LIN {X 0,Y 474.641,Z 374.861,A -85,B 0,C 180,E1 -7413.984,E2 -7413.984} C_VEL
LIN {X 0,Y 474.578,Z 374.865,A -85,B 0,C 180,E1 -7416.9,E2 -7416.9} C_VEL
LIN {X 0,Y 474.63,Z 374.866,A -85,B 0,C 180,E1 -7419.648,E2 -7419.648} C_VEL
LIN {X 0,Y 474.638,Z 374.859,A -85,B 0,C 180,E1 -7422.932,E2 -7422.932} C_VEL
LIN {X 0,Y 474.612,Z 374.864,A -85,B 0,C 180,E1 -7425.895,E2 -7425.895} C_VEL
LIN {X 0,Y 474.63,Z 374.861,A -85,B 0,C 180,E1 -7429.041,E2 -7429.041} C_VEL
LIN {X 0,Y 474.613,Z 374.865,A -85,B 0,C 180,E1 -7431.704,E2 -7431.704} C_VEL
LIN {X 0,Y 474.633,Z 374.859,A -85,B 0,C 180,E1 -7434.726,E2 -7434.726} C_VEL
LIN {X 0,Y 474.638,Z 374.86,A -85,B 0,C 180,E1 -7437.788,E2 -7437.788} C_VEL
LIN {X 0,Y 474.627,Z 374.862,A -85,B 0,C 180,E1 -7440.885,E2 -7440.885} C_VEL
LIN {X 0,Y 474.663,Z 374.859,A -85,B 0,C 180,E1 -7443.629,E2 -7443.629} C_VEL
LIN {X 0,Y 474.638,Z 374.864,A -85,B 0,C 180,E1 -7446.642,E2 -7446.642} C_VEL
LIN {X 0,Y 474.644,Z 374.992,A -85,B 0,C 180,E1 -7447.845,E2 -7447.845} C_VEL
LIN {X 0,Y 475.969,Z 382.275,A -85,B 0,C 180,E1 -7449.471,E2 -7449.471} C_VEL
LIN {X 0,Y 475.834,Z 390.327,A -85,B 0,C 180,E1 -7451.163,E2 -7451.163} C_VEL
LIN {X 0,Y 475.06,Z 393.516,A -85,B 0,C 180,E1 -7451.731,E2 -7451.731} C_VEL
LIN {X 0,Y 472.954,Z 398.571,A -85,B 0,C 180,E1 -7452.388,E2 -7452.388} C_VEL
LIN {X 0,Y 470.99,Z 404.444,A -85,B 0,C 180,E1 -7452.913,E2 -7452.913} C_VEL
LIN {X 0,Y 470.407,Z 409.431,A -85,B 0,C 180,E1 -7453.202,E2 -7453.202} C_VEL
LIN {X 0,Y 470.813,Z 412.936,A -85,B 0,C 180,E1 -7453.324,E2 -7453.324} C_VEL
LIN {X 0,Y 471.386,Z 416.146,A -85,B 0,C 180,E1 -7453.395,E2 -7453.395} C_VEL
LIN {X 0,Y 470.721,Z 508.175,A -85,B 0,C 180,E1 -7454.826,E2 -7454.826} C_VEL
LIN {X 0,Y 470.324,Z 521.294,A -85,B 0,C 180,E1 -7455.201,E2 -7455.201} C_VEL
LIN {X 0,Y 469.941,Z 533.362,A -85,B 0,C 180,E1 -7455.714,E2 -7455.714} C_VEL
LIN {X 0,Y 469.543,Z 544.921,A -85,B 0,C 180,E1 -7456.377,E2 -7456.377} C_VEL
LIN {X 0,Y 469.092,Z 556.415,A -85,B 0,C 180,E1 -7457.233,E2 -7457.233} C_VEL
LIN {X 0,Y 468.56,Z 566.889,A -85,B 0,C 180,E1 -7458.208,E2 -7458.208} C_VEL
LIN {X 0,Y 468.137,Z 575.446,A -85,B 0,C 180,E1 -7459.184,E2 -7459.184} C_VEL
LIN {X 0,Y 467.72,Z 583.328,A -85,B 0,C 180,E1 -7460.268,E2 -7460.268} C_VEL
LIN {X 0,Y 467.35,Z 591.034,A -85,B 0,C 180,E1 -7461.569,E2 -7461.569} C_VEL
LIN {X 0,Y 467.003,Z 598.104,A -85,B 0,C 180,E1 -7463.085,E2 -7463.085} C_VEL
LIN {X 0,Y 466.918,Z 602.812,A -85,B 0,C 180,E1 -7464.385,E2 -7464.385} C_VEL
LIN {X 0,Y 466.744,Z 606.42,A -85,B 0,C 180,E1 -7465.682,E2 -7465.682} C_VEL
LIN {X 0,Y 466.768,Z 608.283,A -85,B 0,C 180,E1 -7466.547,E2 -7466.547} C_VEL
LIN {X 0,Y 466.683,Z 609.689,A -85,B 0,C 180,E1 -7467.411,E2 -7467.411} C_VEL
LIN {X 0,Y 466.62,Z 611.305,A -85,B 0,C 180,E1 -7469.137,E2 -7469.137} C_VEL
LIN {X 0,Y 466.599,Z 611.541,A -85,B 0,C 180,E1 -7470,E2 -7470} C_VEL
LIN {X 0,Y 466.62,Z 611.354,A -85,B 0,C 180,E1 -7470.863,E2 -7470.863} C_VEL
LIN {X 0,Y 466.684,Z 609.803,A -85,B 0,C 180,E1 -7472.59,E2 -7472.59} C_VEL
LIN {X 0,Y 466.767,Z 608.446,A -85,B 0,C 180,E1 -7473.453,E2 -7473.453} C_VEL
LIN {X 0,Y 466.731,Z 605.582,A -85,B 0,C 180,E1 -7474.751,E2 -7474.751} C_VEL
LIN {X 0,Y 466.97,Z 601.692,A -85,B 0,C 180,E1 -7476.048,E2 -7476.048} C_VEL
LIN {X 0,Y 467.099,Z 596.678,A -85,B 0,C 180,E1 -7477.348,E2 -7477.348} C_VEL
LIN {X 0,Y 467.365,Z 590.367,A -85,B 0,C 180,E1 -7478.649,E2 -7478.649} C_VEL
LIN {X 0,Y 467.731,Z 582.464,A -85,B 0,C 180,E1 -7479.951,E2 -7479.951} C_VEL
LIN {X 0,Y 468.241,Z 572.632,A -85,B 0,C 180,E1 -7481.252,E2 -7481.252} C_VEL
LIN {X 0,Y 468.788,Z 562.317,A -85,B 0,C 180,E1 -7482.336,E2 -7482.336} C_VEL
LIN {X 0,Y 469.277,Z 550.683,A -85,B 0,C 180,E1 -7483.312,E2 -7483.312} C_VEL
LIN {X 0,Y 469.761,Z 539.099,A -85,B 0,C 180,E1 -7484.071,E2 -7484.071} C_VEL
LIN {X 0,Y 470.194,Z 527.053,A -85,B 0,C 180,E1 -7484.665,E2 -7484.665} C_VEL
LIN {X 0,Y 470.525,Z 513.933,A -85,B 0,C 180,E1 -7485.125,E2 -7485.125} C_VEL
LIN {X 0,Y 470.775,Z 501.287,A -85,B 0,C 180,E1 -7485.394,E2 -7485.394} C_VEL
LIN {X 0,Y 471.261,Z 415.355,A -85,B 0,C 180,E1 -7486.713,E2 -7486.713} C_VEL
LIN {X 0,Y 468.483,Z 400.834,A -85,B 0,C 180,E1 -7487.055,E2 -7487.055} C_VEL
LIN {X 0,Y 469.089,Z 386.049,A -85,B 0,C 180,E1 -7490.157,E2 -7490.157} C_VEL
LIN {X 0,Y 468.789,Z 381.795,A -85,B 0,C 180,E1 -7491.088,E2 -7491.088} C_VEL
LIN {X 0,Y 467.605,Z 375.744,A -85,B 0,C 180,E1 -7492.478,E2 -7492.478} C_VEL
LIN {X 0,Y 467.614,Z 375.739,A -85,B 0,C 180,E1 -7495.84,E2 -7495.84} C_VEL
LIN {X 0,Y 467.581,Z 375.744,A -85,B 0,C 180,E1 -7498.75,E2 -7498.75} C_VEL
LIN {X 0,Y 467.587,Z 375.736,A -85,B 0,C 180,E1 -7501.74,E2 -7501.74} C_VEL
LIN {X 0,Y 467.57,Z 375.745,A -85,B 0,C 180,E1 -7504.833,E2 -7504.833} C_VEL
LIN {X 0,Y 467.569,Z 375.739,A -85,B 0,C 180,E1 -7508.045,E2 -7508.045} C_VEL
LIN {X 0,Y 467.582,Z 375.737,A -85,B 0,C 180,E1 -7511.277,E2 -7511.277} C_VEL
LIN {X 0,Y 467.558,Z 375.74,A -85,B 0,C 180,E1 -7513.821,E2 -7513.821} C_VEL
LIN {X 0,Y 467.574,Z 375.742,A -85,B 0,C 180,E1 -7516.257,E2 -7516.257} C_VEL
LIN {X 0,Y 467.586,Z 375.741,A -85,B 0,C 180,E1 -7518.723,E2 -7518.723} C_VEL
LIN {X 0,Y 467.569,Z 375.74,A -85,B 0,C 180,E1 -7521.956,E2 -7521.956} C_VEL
LIN {X 0,Y 467.568,Z 375.738,A -85,B 0,C 180,E1 -7525.168,E2 -7525.168} C_VEL
LIN {X 0,Y 467.588,Z 375.743,A -85,B 0,C 180,E1 -7528.26,E2 -7528.26} C_VEL
LIN {X 0,Y 467.582,Z 375.736,A -85,B 0,C 180,E1 -7531.251,E2 -7531.251} C_VEL
LIN {X 0,Y 467.618,Z 375.732,A -85,B 0,C 180,E1 -7533.2,E2 -7533.2} C_VEL
LIN {X 0,Y 467.596,Z 375.739,A -85,B 0,C 180,E1 -7536.469,E2 -7536.469} C_VEL
LIN {X 0,Y 467.63,Z 375.734,A -85,B 0,C 180,E1 -7539.777,E2 -7539.777} C_VEL
LIN {X 0,Y 467.615,Z 375.735,A -85,B 0,C 180,E1 -7542.507,E2 -7542.507} C_VEL
LIN {X 0,Y 467.612,Z 375.733,A -85,B 0,C 180,E1 -7545.197,E2 -7545.197} C_VEL
LIN {X 0,Y 467.662,Z 375.732,A -85,B 0,C 180,E1 -7547.855,E2 -7547.855} C_VEL
LIN {X 0,Y 467.686,Z 375.725,A -85,B 0,C 180,E1 -7551.357,E2 -7551.357} C_VEL
LIN {X 0,Y 467.749,Z 375.723,A -85,B 0,C 180,E1 -7553.963,E2 -7553.963} C_VEL
LIN {X 0,Y 467.865,Z 375.704,A -85,B 0,C 180,E1 -7557.417,E2 -7557.417} C_VEL
LIN {X 0,Y 467.888,Z 375.704,A -85,B 0,C 180,E1 -7560,E2 -7560} C_VEL
LIN {X 0,Y 467.865,Z 375.701,A -85,B 0,C 180,E1 -7562.583,E2 -7562.583} C_VEL
LIN {X 0,Y 467.748,Z 375.72,A -85,B 0,C 180,E1 -7566.037,E2 -7566.037} C_VEL
LIN {X 0,Y 467.674,Z 375.725,A -85,B 0,C 180,E1 -7568.643,E2 -7568.643} C_VEL
LIN {X 0,Y 467.689,Z 375.725,A -85,B 0,C 180,E1 -7572.145,E2 -7572.145} C_VEL
LIN {X 0,Y 467.655,Z 375.731,A -85,B 0,C 180,E1 -7575.885,E2 -7575.885} C_VEL
LIN {X 0,Y 467.629,Z 375.736,A -85,B 0,C 180,E1 -7579.308,E2 -7579.308} C_VEL
LIN {X 0,Y 467.539,Z 375.743,A -85,B 0,C 180,E1 -7582.074,E2 -7582.074} C_VEL
LIN {X 0,Y 467.59,Z 375.737,A -85,B 0,C 180,E1 -7584.888,E2 -7584.888} C_VEL
LIN {X 0,Y 467.625,Z 375.734,A -85,B 0,C 180,E1 -7587.769,E2 -7587.769} C_VEL
LIN {X 0,Y 467.572,Z 375.742,A -85,B 0,C 180,E1 -7591.045,E2 -7591.045} C_VEL
LIN {X 0,Y 467.581,Z 375.736,A -85,B 0,C 180,E1 -7594.24,E2 -7594.24} C_VEL
LIN {X 0,Y 467.552,Z 375.748,A -85,B 0,C 180,E1 -7597.186,E2 -7597.186} C_VEL
LIN {X 0,Y 467.578,Z 375.737,A -85,B 0,C 180,E1 -7600.265,E2 -7600.265} C_VEL
LIN {X 0,Y 467.59,Z 375.737,A -85,B 0,C 180,E1 -7602.567,E2 -7602.567} C_VEL
LIN {X 0,Y 467.575,Z 375.745,A -85,B 0,C 180,E1 -7605.053,E2 -7605.053} C_VEL
LIN {X 0,Y 467.592,Z 375.738,A -85,B 0,C 180,E1 -7607.44,E2 -7607.44} C_VEL
LIN {X 0,Y 467.586,Z 375.742,A -85,B 0,C 180,E1 -7610.855,E2 -7610.855} C_VEL
LIN {X 0,Y 467.564,Z 375.739,A -85,B 0,C 180,E1 -7614.261,E2 -7614.261} C_VEL
LIN {X 0,Y 467.585,Z 375.739,A -85,B 0,C 180,E1 -7617.321,E2 -7617.321} C_VEL
LIN {X 0,Y 467.574,Z 375.745,A -85,B 0,C 180,E1 -7620.667,E2 -7620.667} C_VEL
LIN {X 0,Y 467.62,Z 375.738,A -85,B 0,C 180,E1 -7623.2,E2 -7623.2} C_VEL
LIN {X 0,Y 467.656,Z 375.805,A -85,B 0,C 180,E1 -7624.532,E2 -7624.532} C_VEL
LIN {X 0,Y 469.817,Z 387.641,A -85,B 0,C 180,E1 -7626.879,E2 -7626.879} C_VEL
LIN {X 0,Y 469.192,Z 401.354,A -85,B 0,C 180,E1 -7629.39,E2 -7629.39} C_VEL
LIN {X 0,Y 468.532,Z 417.506,A -85,B 0,C 180,E1 -7632.317,E2 -7632.317} C_VEL
LIN {X 0,Y 468.356,Z 421.166,A -85,B 0,C 180,E1 -7632.978,E2 -7632.978} C_VEL
LIN {X 0,Y 471.298,Z 439.48,A -85,B 0,C 180,E1 -7633.378,E2 -7633.378} C_VEL
LIN {X 0,Y 470.596,Z 529.173,A -85,B 0,C 180,E1 -7634.766,E2 -7634.766} C_VEL
LIN {X 0,Y 470.239,Z 542.449,A -85,B 0,C 180,E1 -7635.143,E2 -7635.143} C_VEL
LIN {X 0,Y 469.768,Z 554.613,A -85,B 0,C 180,E1 -7635.653,E2 -7635.653} C_VEL
LIN {X 0,Y 469.294,Z 566.886,A -85,B 0,C 180,E1 -7636.357,E2 -7636.357} C_VEL
LIN {X 0,Y 468.767,Z 578.482,A -85,B 0,C 180,E1 -7637.224,E2 -7637.224} C_VEL
LIN {X 0,Y 468.291,Z 588.923,A -85,B 0,C 180,E1 -7638.201,E2 -7638.201} C_VEL
LIN {X 0,Y 467.866,Z 597.459,A -85,B 0,C 180,E1 -7639.177,E2 -7639.177} C_VEL
LIN {X 0,Y 467.468,Z 605.335,A -85,B 0,C 180,E1 -7640.262,E2 -7640.262} C_VEL
LIN {X 0,Y 467.123,Z 613.026,A -85,B 0,C 180,E1 -7641.565,E2 -7641.565} C_VEL
LIN {X 0,Y 466.86,Z 620.118,A -85,B 0,C 180,E1 -7643.083,E2 -7643.083} C_VEL
LIN {X 0,Y 466.784,Z 624.837,A -85,B 0,C 180,E1 -7644.384,E2 -7644.384} C_VEL
LIN {X 0,Y 466.647,Z 628.44,A -85,B 0,C 180,E1 -7645.681,E2 -7645.681} C_VEL
LIN {X 0,Y 466.661,Z 630.3,A -85,B 0,C 180,E1 -7646.546,E2 -7646.546} C_VEL
LIN {X 0,Y 466.66,Z 631.695,A -85,B 0,C 180,E1 -7647.41,E2 -7647.41} C_VEL
LIN {X 0,Y 466.589,Z 633.296,A -85,B 0,C 180,E1 -7649.137,E2 -7649.137} C_VEL
LIN {X 0,Y 466.598,Z 633.513,A -85,B 0,C 180,E1 -7650,E2 -7650} C_VEL
LIN {X 0,Y 466.607,Z 632.691,A -85,B 0,C 180,E1 -7651.726,E2 -7651.726} C_VEL
LIN {X 0,Y 466.66,Z 631.698,A -85,B 0,C 180,E1 -7652.589,E2 -7652.589} C_VEL
LIN {X 0,Y 466.661,Z 630.304,A -85,B 0,C 180,E1 -7653.453,E2 -7653.453} C_VEL
LIN {X 0,Y 466.692,Z 627.372,A -85,B 0,C 180,E1 -7654.751,E2 -7654.751} C_VEL
LIN {X 0,Y 466.779,Z 623.403,A -85,B 0,C 180,E1 -7656.05,E2 -7656.05} C_VEL
LIN {X 0,Y 466.978,Z 617.299,A -85,B 0,C 180,E1 -7657.567,E2 -7657.567} C_VEL
LIN {X 0,Y 467.232,Z 610.628,A -85,B 0,C 180,E1 -7658.869,E2 -7658.869} C_VEL
LIN {X 0,Y 467.59,Z 602.351,A -85,B 0,C 180,E1 -7660.172,E2 -7660.172} C_VEL
LIN {X 0,Y 468.057,Z 593.87,A -85,B 0,C 180,E1 -7661.256,E2 -7661.256} C_VEL
LIN {X 0,Y 468.583,Z 583.778,A -85,B 0,C 180,E1 -7662.304,E2 -7662.304} C_VEL
LIN {X 0,Y 468.97,Z 573.014,A -85,B 0,C 180,E1 -7663.211,E2 -7663.211} C_VEL
LIN {X 0,Y 469.484,Z 561.645,A -85,B 0,C 180,E1 -7663.968,E2 -7663.968} C_VEL
LIN {X 0,Y 469.931,Z 549.982,A -85,B 0,C 180,E1 -7664.563,E2 -7664.563} C_VEL
LIN {X 0,Y 470.365,Z 537.457,A -85,B 0,C 180,E1 -7665.019,E2 -7665.019} C_VEL
LIN {X 0,Y 470.637,Z 524.776,A -85,B 0,C 180,E1 -7665.315,E2 -7665.315} C_VEL
LIN {X 0,Y 471.121,Z 438.262,A -85,B 0,C 180,E1 -7666.646,E2 -7666.646} C_VEL
LIN {X 0,Y 468.379,Z 421.186,A -85,B 0,C 180,E1 -7667.014,E2 -7667.014} C_VEL
LIN {X 0,Y 469.104,Z 403.829,A -85,B 0,C 180,E1 -7670.156,E2 -7670.156} C_VEL
LIN {X 0,Y 469.829,Z 388.878,A -85,B 0,C 180,E1 -7672.888,E2 -7672.888} C_VEL
LIN {X 0,Y 469.111,Z 383.371,A -85,B 0,C 180,E1 -7673.953,E2 -7673.953} C_VEL
LIN {X 0,Y 467.646,Z 375.734,A -85,B 0,C 180,E1 -7675.52,E2 -7675.52} C_VEL
LIN {X 0,Y 467.63,Z 375.736,A -85,B 0,C 180,E1 -7677.768,E2 -7677.768} C_VEL
LIN {X 0,Y 467.572,Z 375.745,A -85,B 0,C 180,E1 -7681.045,E2 -7681.045} C_VEL
LIN {X 0,Y 467.591,Z 375.735,A -85,B 0,C 180,E1 -7684.242,E2 -7684.242} C_VEL
LIN {X 0,Y 467.55,Z 375.746,A -85,B 0,C 180,E1 -7687.186,E2 -7687.186} C_VEL
LIN {X 0,Y 467.579,Z 375.737,A -85,B 0,C 180,E1 -7690.264,E2 -7690.264} C_VEL
LIN {X 0,Y 467.588,Z 375.739,A -85,B 0,C 180,E1 -7692.567,E2 -7692.567} C_VEL
LIN {X 0,Y 467.573,Z 375.744,A -85,B 0,C 180,E1 -7695.053,E2 -7695.053} C_VEL
LIN {X 0,Y 467.591,Z 375.737,A -85,B 0,C 180,E1 -7697.44,E2 -7697.44} C_VEL
LIN {X 0,Y 467.584,Z 375.744,A -85,B 0,C 180,E1 -7700.855,E2 -7700.855} C_VEL
LIN {X 0,Y 467.562,Z 375.741,A -85,B 0,C 180,E1 -7704.261,E2 -7704.261} C_VEL
LIN {X 0,Y 467.584,Z 375.737,A -85,B 0,C 180,E1 -7707.321,E2 -7707.321} C_VEL
LIN {X 0,Y 467.573,Z 375.746,A -85,B 0,C 180,E1 -7710.667,E2 -7710.667} C_VEL
LIN {X 0,Y 467.615,Z 375.734,A -85,B 0,C 180,E1 -7713.2,E2 -7713.2} C_VEL
LIN {X 0,Y 467.593,Z 375.742,A -85,B 0,C 180,E1 -7716.469,E2 -7716.469} C_VEL
LIN {X 0,Y 467.627,Z 375.731,A -85,B 0,C 180,E1 -7719.777,E2 -7719.777} C_VEL
LIN {X 0,Y 467.61,Z 375.741,A -85,B 0,C 180,E1 -7722.507,E2 -7722.507} C_VEL
LIN {X 0,Y 467.609,Z 375.733,A -85,B 0,C 180,E1 -7725.197,E2 -7725.197} C_VEL
LIN {X 0,Y 467.686,Z 375.725,A -85,B 0,C 180,E1 -7727.855,E2 -7727.855} C_VEL
LIN {X 0,Y 467.673,Z 375.725,A -85,B 0,C 180,E1 -7731.357,E2 -7731.357} C_VEL
LIN {X 0,Y 467.74,Z 375.72,A -85,B 0,C 180,E1 -7733.963,E2 -7733.963} C_VEL
LIN {X 0,Y 467.862,Z 375.702,A -85,B 0,C 180,E1 -7737.417,E2 -7737.417} C_VEL
LIN {X 0,Y 467.886,Z 375.704,A -85,B 0,C 180,E1 -7740,E2 -7740} C_VEL
LIN {X 0,Y 467.863,Z 375.704,A -85,B 0,C 180,E1 -7742.583,E2 -7742.583} C_VEL
LIN {X 0,Y 467.747,Z 375.723,A -85,B 0,C 180,E1 -7746.037,E2 -7746.037} C_VEL
LIN {X 0,Y 467.683,Z 375.725,A -85,B 0,C 180,E1 -7748.643,E2 -7748.643} C_VEL
LIN {X 0,Y 467.659,Z 375.733,A -85,B 0,C 180,E1 -7752.145,E2 -7752.145} C_VEL
LIN {X 0,Y 467.642,Z 375.733,A -85,B 0,C 180,E1 -7755.695,E2 -7755.695} C_VEL
LIN {X 0,Y 467.621,Z 375.732,A -85,B 0,C 180,E1 -7758.765,E2 -7758.765} C_VEL
LIN {X 0,Y 467.584,Z 375.737,A -85,B 0,C 180,E1 -7761.269,E2 -7761.269} C_VEL
LIN {X 0,Y 467.577,Z 375.744,A -85,B 0,C 180,E1 -7763.943,E2 -7763.943} C_VEL
LIN {X 0,Y 467.619,Z 375.732,A -85,B 0,C 180,E1 -7766.8,E2 -7766.8} C_VEL
LIN {X 0,Y 467.583,Z 375.744,A -85,B 0,C 180,E1 -7769.736,E2 -7769.736} C_VEL
LIN {X 0,Y 467.586,Z 375.736,A -85,B 0,C 180,E1 -7772.758,E2 -7772.758} C_VEL
LIN {X 0,Y 467.559,Z 375.744,A -85,B 0,C 180,E1 -7775.889,E2 -7775.889} C_VEL
LIN {X 0,Y 467.585,Z 375.738,A -85,B 0,C 180,E1 -7779.145,E2 -7779.145} C_VEL
LIN {X 0,Y 467.589,Z 375.735,A -85,B 0,C 180,E1 -7782.567,E2 -7782.567} C_VEL
LIN {X 0,Y 467.573,Z 375.74,A -85,B 0,C 180,E1 -7785.053,E2 -7785.053} C_VEL
LIN {X 0,Y 467.591,Z 375.743,A -85,B 0,C 180,E1 -7787.44,E2 -7787.44} C_VEL
LIN {X 0,Y 467.585,Z 375.737,A -85,B 0,C 180,E1 -7790.855,E2 -7790.855} C_VEL
LIN {X 0,Y 467.566,Z 375.738,A -85,B 0,C 180,E1 -7794.26,E2 -7794.26} C_VEL
LIN {X 0,Y 467.584,Z 375.744,A -85,B 0,C 180,E1 -7797.321,E2 -7797.321} C_VEL
LIN {X 0,Y 467.573,Z 375.739,A -85,B 0,C 180,E1 -7800.667,E2 -7800.667} C_VEL
LIN {X 0,Y 467.62,Z 375.74,A -85,B 0,C 180,E1 -7803.2,E2 -7803.2} C_VEL
LIN {X 0,Y 467.595,Z 375.741,A -85,B 0,C 180,E1 -7806.468,E2 -7806.468} C_VEL
LIN {X 0,Y 467.605,Z 375.794,A -85,B 0,C 180,E1 -7807.639,E2 -7807.639} C_VEL
LIN {X 0,Y 469.003,Z 383.485,A -85,B 0,C 180,E1 -7809.381,E2 -7809.381} C_VEL
LIN {X 0,Y 468.876,Z 391.333,A -85,B 0,C 180,E1 -7811.055,E2 -7811.055} C_VEL
LIN {X 0,Y 468.462,Z 400.892,A -85,B 0,C 180,E1 -7813.045,E2 -7813.045} C_VEL
LIN {X 0,Y 470.813,Z 412.936,A -85,B 0,C 180,E1 -7813.324,E2 -7813.324} C_VEL
LIN {X 0,Y 471.197,Z 416.752,A -85,B 0,C 180,E1 -7813.398,E2 -7813.398} C_VEL
LIN {X 0,Y 470.793,Z 420.616,A -85,B 0,C 180,E1 -7813.443,E2 -7813.443} C_VEL
LIN {X 0,Y 468.576,Z 428.234,A -85,B 0,C 180,E1 -7813.481,E2 -7813.481} C_VEL
LIN {X 0,Y 465.278,Z 437.865,A -85,B 0,C 180,E1 -7813.511,E2 -7813.511} C_VEL
LIN {X 0,Y 464.375,Z 443.823,A -85,B 0,C 180,E1 -7813.572,E2 -7813.572} C_VEL
LIN {X 0,Y 463.889,Z 508.36,A -85,B 0,C 180,E1 -7814.597,E2 -7814.597} C_VEL
LIN {X 0,Y 463.476,Z 521.474,A -85,B 0,C 180,E1 -7814.977,E2 -7814.977} C_VEL
LIN {X 0,Y 463.074,Z 533.538,A -85,B 0,C 180,E1 -7815.498,E2 -7815.498} C_VEL
LIN {X 0,Y 462.663,Z 544.918,A -85,B 0,C 180,E1 -7816.158,E2 -7816.158} C_VEL
LIN {X 0,Y 462.18,Z 556.588,A -85,B 0,C 180,E1 -7817.039,E2 -7817.039} C_VEL
LIN {X 0,Y 461.625,Z 567.06,A -85,B 0,C 180,E1 -7818.028,E2 -7818.028} C_VEL
LIN {X 0,Y 461.142,Z 575.618,A -85,B 0,C 180,E1 -7819.018,E2 -7819.018} C_VEL
LIN {X 0,Y 460.724,Z 583.498,A -85,B 0,C 180,E1 -7820.119,E2 -7820.119} C_VEL
LIN {X 0,Y 460.305,Z 591.204,A -85,B 0,C 180,E1 -7821.439,E2 -7821.439} C_VEL
LIN {X 0,Y 459.946,Z 598.273,A -85,B 0,C 180,E1 -7822.979,E2 -7822.979} C_VEL
LIN {X 0,Y 459.865,Z 602.98,A -85,B 0,C 180,E1 -7824.299,E2 -7824.299} C_VEL
LIN {X 0,Y 459.651,Z 606.589,A -85,B 0,C 180,E1 -7825.616,E2 -7825.616} C_VEL
LIN {X 0,Y 459.682,Z 608.451,A -85,B 0,C 180,E1 -7826.494,E2 -7826.494} C_VEL
LIN {X 0,Y 459.607,Z 609.857,A -85,B 0,C 180,E1 -7827.371,E2 -7827.371} C_VEL
LIN {X 0,Y 459.523,Z 611.472,A -85,B 0,C 180,E1 -7829.124,E2 -7829.124} C_VEL
LIN {X 0,Y 459.501,Z 611.708,A -85,B 0,C 180,E1 -7830,E2 -7830} C_VEL
LIN {X 0,Y 459.523,Z 611.521,A -85,B 0,C 180,E1 -7830.876,E2 -7830.876} C_VEL
LIN {X 0,Y 459.607,Z 609.969,A -85,B 0,C 180,E1 -7832.629,E2 -7832.629} C_VEL
LIN {X 0,Y 459.681,Z 608.612,A -85,B 0,C 180,E1 -7833.506,E2 -7833.506} C_VEL
LIN {X 0,Y 459.659,Z 605.748,A -85,B 0,C 180,E1 -7834.824,E2 -7834.824} C_VEL
LIN {X 0,Y 459.903,Z 601.858,A -85,B 0,C 180,E1 -7836.141,E2 -7836.141} C_VEL
LIN {X 0,Y 460.048,Z 596.844,A -85,B 0,C 180,E1 -7837.461,E2 -7837.461} C_VEL
LIN {X 0,Y 460.348,Z 590.531,A -85,B 0,C 180,E1 -7838.782,E2 -7838.782} C_VEL
LIN {X 0,Y 460.725,Z 582.628,A -85,B 0,C 180,E1 -7840.104,E2 -7840.104} C_VEL
LIN {X 0,Y 461.28,Z 572.795,A -85,B 0,C 180,E1 -7841.424,E2 -7841.424} C_VEL
LIN {X 0,Y 461.84,Z 562.523,A -85,B 0,C 180,E1 -7842.52,E2 -7842.52} C_VEL
LIN {X 0,Y 462.341,Z 551.523,A -85,B 0,C 180,E1 -7843.462,E2 -7843.462} C_VEL
LIN {X 0,Y 462.83,Z 541.082,A -85,B 0,C 180,E1 -7844.174,E2 -7844.174} C_VEL
LIN {X 0,Y 463.245,Z 529.745,A -85,B 0,C 180,E1 -7844.778,E2 -7844.778} C_VEL
LIN {X 0,Y 463.629,Z 516.828,A -85,B 0,C 180,E1 -7845.271,E2 -7845.271} C_VEL
LIN {X 0,Y 463.918,Z 503.032,A -85,B 0,C 180,E1 -7845.599,E2 -7845.599} C_VEL
LIN {X 0,Y 464.453,Z 416.258,A -85,B 0,C 180,E1 -7846.953,E2 -7846.953} C_VEL
LIN {X 0,Y 461.535,Z 400.995,A -85,B 0,C 180,E1 -7847.32,E2 -7847.32} C_VEL
LIN {X 0,Y 462.146,Z 387.258,A -85,B 0,C 180,E1 -7850.241,E2 -7850.241} C_VEL
LIN {X 0,Y 461.793,Z 383,A -85,B 0,C 180,E1 -7851.19,E2 -7851.19} C_VEL
LIN {X 0,Y 460.543,Z 376.624,A -85,B 0,C 180,E1 -7852.664,E2 -7852.664} C_VEL
LIN {X 0,Y 460.572,Z 376.617,A -85,B 0,C 180,E1 -7855.802,E2 -7855.802} C_VEL
LIN {X 0,Y 460.557,Z 376.613,A -85,B 0,C 180,E1 -7858.233,E2 -7858.233} C_VEL
LIN {X 0,Y 460.525,Z 376.617,A -85,B 0,C 180,E1 -7861.283,E2 -7861.283} C_VEL
LIN {X 0,Y 460.536,Z 376.619,A -85,B 0,C 180,E1 -7864.506,E2 -7864.506} C_VEL
LIN {X 0,Y 460.505,Z 376.618,A -85,B 0,C 180,E1 -7867.623,E2 -7867.623} C_VEL
LIN {X 0,Y 460.543,Z 376.617,A -85,B 0,C 180,E1 -7870.269,E2 -7870.269} C_VEL
LIN {X 0,Y 460.504,Z 376.618,A -85,B 0,C 180,E1 -7873.375,E2 -7873.375} C_VEL
LIN {X 0,Y 460.514,Z 376.624,A -85,B 0,C 180,E1 -7876.626,E2 -7876.626} C_VEL
LIN {X 0,Y 460.547,Z 376.613,A -85,B 0,C 180,E1 -7879.731,E2 -7879.731} C_VEL
LIN {X 0,Y 460.53,Z 376.622,A -85,B 0,C 180,E1 -7882.52,E2 -7882.52} C_VEL
LIN {X 0,Y 460.55,Z 376.613,A -85,B 0,C 180,E1 -7885.624,E2 -7885.624} C_VEL
LIN {X 0,Y 460.542,Z 376.616,A -85,B 0,C 180,E1 -7888.745,E2 -7888.745} C_VEL
LIN {X 0,Y 460.594,Z 376.615,A -85,B 0,C 180,E1 -7892.252,E2 -7892.252} C_VEL
LIN {X 0,Y 460.536,Z 376.616,A -85,B 0,C 180,E1 -7895.667,E2 -7895.667} C_VEL
LIN {X 0,Y 460.526,Z 376.618,A -85,B 0,C 180,E1 -7898.578,E2 -7898.578} C_VEL
LIN {X 0,Y 460.596,Z 376.607,A -85,B 0,C 180,E1 -7901.311,E2 -7901.311} C_VEL
LIN {X 0,Y 460.609,Z 376.613,A -85,B 0,C 180,E1 -7904.059,E2 -7904.059} C_VEL
LIN {X 0,Y 460.615,Z 376.608,A -85,B 0,C 180,E1 -7907.666,E2 -7907.666} C_VEL
LIN {X 0,Y 460.633,Z 376.602,A -85,B 0,C 180,E1 -7911.224,E2 -7911.224} C_VEL
LIN {X 0,Y 460.716,Z 376.599,A -85,B 0,C 180,E1 -7913.87,E2 -7913.87} C_VEL
LIN {X 0,Y 460.806,Z 376.583,A -85,B 0,C 180,E1 -7917.377,E2 -7917.377} C_VEL
LIN {X 0,Y 460.858,Z 376.58,A -85,B 0,C 180,E1 -7920,E2 -7920} C_VEL
LIN {X 0,Y 460.806,Z 376.581,A -85,B 0,C 180,E1 -7922.622,E2 -7922.622} C_VEL
LIN {X 0,Y 460.713,Z 376.595,A -85,B 0,C 180,E1 -7926.13,E2 -7926.13} C_VEL
LIN {X 0,Y 460.624,Z 376.603,A -85,B 0,C 180,E1 -7928.776,E2 -7928.776} C_VEL
LIN {X 0,Y 460.64,Z 376.601,A -85,B 0,C 180,E1 -7932.457,E2 -7932.457} C_VEL
LIN {X 0,Y 460.605,Z 376.608,A -85,B 0,C 180,E1 -7935.997,E2 -7935.997} C_VEL
LIN {X 0,Y 460.576,Z 376.61,A -85,B 0,C 180,E1 -7938.902,E2 -7938.902} C_VEL
LIN {X 0,Y 460.521,Z 376.624,A -85,B 0,C 180,E1 -7941.485,E2 -7941.485} C_VEL
LIN {X 0,Y 460.536,Z 376.614,A -85,B 0,C 180,E1 -7944.333,E2 -7944.333} C_VEL
LIN {X 0,Y 460.576,Z 376.615,A -85,B 0,C 180,E1 -7947.244,E2 -7947.244} C_VEL
LIN {X 0,Y 460.515,Z 376.617,A -85,B 0,C 180,E1 -7950.24,E2 -7950.24} C_VEL
LIN {X 0,Y 460.524,Z 376.623,A -85,B 0,C 180,E1 -7953.325,E2 -7953.325} C_VEL
LIN {X 0,Y 460.48,Z 376.622,A -85,B 0,C 180,E1 -7956.529,E2 -7956.529} C_VEL
LIN {X 0,Y 460.531,Z 376.616,A -85,B 0,C 180,E1 -7959.863,E2 -7959.863} C_VEL
LIN {X 0,Y 460.521,Z 376.621,A -85,B 0,C 180,E1 -7962.901,E2 -7962.901} C_VEL
LIN {X 0,Y 460.515,Z 376.617,A -85,B 0,C 180,E1 -7965.83,E2 -7965.83} C_VEL
LIN {X 0,Y 460.534,Z 376.622,A -85,B 0,C 180,E1 -7968.989,E2 -7968.989} C_VEL
LIN {X 0,Y 460.53,Z 376.619,A -85,B 0,C 180,E1 -7971.267,E2 -7971.267} C_VEL
LIN {X 0,Y 460.515,Z 376.62,A -85,B 0,C 180,E1 -7974.554,E2 -7974.554} C_VEL
LIN {X 0,Y 460.535,Z 376.614,A -85,B 0,C 180,E1 -7977.715,E2 -7977.715} C_VEL
LIN {X 0,Y 460.544,Z 376.621,A -85,B 0,C 180,E1 -7980.769,E2 -7980.769} C_VEL
LIN {X 0,Y 460.567,Z 376.616,A -85,B 0,C 180,E1 -7983.735,E2 -7983.735} C_VEL
LIN {X 0,Y 460.6,Z 376.811,A -85,B 0,C 180,E1 -7984.337,E2 -7984.337} C_VEL
LIN {X 0,Y 462.712,Z 387.553,A -85,B 0,C 180,E1 -7986.513,E2 -7986.513} C_VEL
LIN {X 0,Y 462.755,Z 392.484,A -85,B 0,C 180,E1 -7987.45,E2 -7987.45} C_VEL
LIN {X 0,Y 461.836,Z 411.614,A -85,B 0,C 180,E1 -7990.989,E2 -7990.989} C_VEL
LIN {X 0,Y 461.385,Z 421.061,A -85,B 0,C 180,E1 -7992.72,E2 -7992.72} C_VEL
LIN {X 0,Y 464.478,Z 439.985,A -85,B 0,C 180,E1 -7993.137,E2 -7993.137} C_VEL
LIN {X 0,Y 463.762,Z 529.016,A -85,B 0,C 180,E1 -7994.536,E2 -7994.536} C_VEL
LIN {X 0,Y 463.386,Z 542.289,A -85,B 0,C 180,E1 -7994.918,E2 -7994.918} C_VEL
LIN {X 0,Y 462.902,Z 554.451,A -85,B 0,C 180,E1 -7995.436,E2 -7995.436} C_VEL
LIN {X 0,Y 462.398,Z 566.722,A -85,B 0,C 180,E1 -7996.15,E2 -7996.15} C_VEL
LIN {X 0,Y 461.777,Z 578.316,A -85,B 0,C 180,E1 -7997.027,E2 -7997.027} C_VEL
LIN {X 0,Y 461.334,Z 588.758,A -85,B 0,C 180,E1 -7998.02,E2 -7998.02} C_VEL
LIN {X 0,Y 460.848,Z 597.293,A -85,B 0,C 180,E1 -7999.01,E2 -7999.01} C_VEL
LIN {X 0,Y 460.454,Z 605.168,A -85,B 0,C 180,E1 -8000.112,E2 -8000.112} C_VEL
LIN {X 0,Y 460.057,Z 612.859,A -85,B 0,C 180,E1 -8001.434,E2 -8001.434} C_VEL
LIN {X 0,Y 459.78,Z 619.951,A -85,B 0,C 180,E1 -8002.976,E2 -8002.976} C_VEL
LIN {X 0,Y 459.683,Z 624.669,A -85,B 0,C 180,E1 -8004.296,E2 -8004.296} C_VEL
LIN {X 0,Y 459.565,Z 628.273,A -85,B 0,C 180,E1 -8005.614,E2 -8005.614} C_VEL
LIN {X 0,Y 459.557,Z 630.133,A -85,B 0,C 180,E1 -8006.493,E2 -8006.493} C_VEL
LIN {X 0,Y 459.581,Z 631.528,A -85,B 0,C 180,E1 -8007.37,E2 -8007.37} C_VEL
LIN {X 0,Y 459.495,Z 633.129,A -85,B 0,C 180,E1 -8009.123,E2 -8009.123} C_VEL
LIN {X 0,Y 459.501,Z 633.346,A -85,B 0,C 180,E1 -8010,E2 -8010} C_VEL
LIN {X 0,Y 459.52,Z 632.524,A -85,B 0,C 180,E1 -8011.753,E2 -8011.753} C_VEL
LIN {X 0,Y 459.581,Z 631.531,A -85,B 0,C 180,E1 -8012.629,E2 -8012.629} C_VEL
LIN {X 0,Y 459.557,Z 630.136,A -85,B 0,C 180,E1 -8013.507,E2 -8013.507} C_VEL
LIN {X 0,Y 459.623,Z 627.204,A -85,B 0,C 180,E1 -8014.824,E2 -8014.824} C_VEL
LIN {X 0,Y 459.714,Z 622.205,A -85,B 0,C 180,E1 -8016.431,E2 -8016.431} C_VEL
LIN {X 0,Y 459.95,Z 616.119,A -85,B 0,C 180,E1 -8017.904,E2 -8017.904} C_VEL
LIN {X 0,Y 460.232,Z 609.222,A -85,B 0,C 180,E1 -8019.227,E2 -8019.227} C_VEL
LIN {X 0,Y 460.636,Z 600.595,A -85,B 0,C 180,E1 -8020.549,E2 -8020.549} C_VEL
LIN {X 0,Y 461.206,Z 591.751,A -85,B 0,C 180,E1 -8021.648,E2 -8021.648} C_VEL
LIN {X 0,Y 461.67,Z 582.034,A -85,B 0,C 180,E1 -8022.641,E2 -8022.641} C_VEL
LIN {X 0,Y 462.123,Z 571.415,A -85,B 0,C 180,E1 -8023.522,E2 -8023.522} C_VEL
LIN {X 0,Y 462.645,Z 559.55,A -85,B 0,C 180,E1 -8024.291,E2 -8024.291} C_VEL
LIN {X 0,Y 463.206,Z 547.207,A -85,B 0,C 180,E1 -8024.891,E2 -8024.891} C_VEL
LIN {X 0,Y 463.58,Z 534.535,A -85,B 0,C 180,E1 -8025.329,E2 -8025.329} C_VEL
LIN {X 0,Y 463.887,Z 521.297,A -85,B 0,C 180,E1 -8025.6,E2 -8025.6} C_VEL
LIN {X 0,Y 464.342,Z 439.269,A -85,B 0,C 180,E1 -8026.877,E2 -8026.877} C_VEL
LIN {X 0,Y 461.399,Z 420.95,A -85,B 0,C 180,E1 -8027.292,E2 -8027.292} C_VEL
LIN {X 0,Y 462.141,Z 404.92,A -85,B 0,C 180,E1 -8030.241,E2 -8030.241} C_VEL
LIN {X 0,Y 462.898,Z 389.98,A -85,B 0,C 180,E1 -8033.014,E2 -8033.014} C_VEL
LIN {X 0,Y 462.001,Z 383.721,A -85,B 0,C 180,E1 -8034.25,E2 -8034.25} C_VEL
LIN {X 0,Y 460.594,Z 376.612,A -85,B 0,C 180,E1 -8035.711,E2 -8035.711} C_VEL
LIN {X 0,Y 460.558,Z 376.616,A -85,B 0,C 180,E1 -8038.233,E2 -8038.233} C_VEL
LIN {X 0,Y 460.525,Z 376.621,A -85,B 0,C 180,E1 -8041.283,E2 -8041.283} C_VEL
LIN {X 0,Y 460.534,Z 376.616,A -85,B 0,C 180,E1 -8044.506,E2 -8044.506} C_VEL
LIN {X 0,Y 460.503,Z 376.619,A -85,B 0,C 180,E1 -8047.623,E2 -8047.623} C_VEL
LIN {X 0,Y 460.544,Z 376.614,A -85,B 0,C 180,E1 -8050.269,E2 -8050.269} C_VEL
LIN {X 0,Y 460.502,Z 376.621,A -85,B 0,C 180,E1 -8053.375,E2 -8053.375} C_VEL
LIN {X 0,Y 460.511,Z 376.622,A -85,B 0,C 180,E1 -8056.626,E2 -8056.626} C_VEL
LIN {X 0,Y 460.545,Z 376.613,A -85,B 0,C 180,E1 -8059.73,E2 -8059.73} C_VEL
LIN {X 0,Y 460.501,Z 376.623,A -85,B 0,C 180,E1 -8062.524,E2 -8062.524} C_VEL
LIN {X 0,Y 460.548,Z 376.613,A -85,B 0,C 180,E1 -8065.624,E2 -8065.624} C_VEL
LIN {X 0,Y 460.539,Z 376.621,A -85,B 0,C 180,E1 -8068.745,E2 -8068.745} C_VEL
LIN {X 0,Y 460.591,Z 376.61,A -85,B 0,C 180,E1 -8072.252,E2 -8072.252} C_VEL
LIN {X 0,Y 460.533,Z 376.614,A -85,B 0,C 180,E1 -8075.667,E2 -8075.667} C_VEL
LIN {X 0,Y 460.524,Z 376.623,A -85,B 0,C 180,E1 -8078.578,E2 -8078.578} C_VEL
LIN {X 0,Y 460.594,Z 376.607,A -85,B 0,C 180,E1 -8081.311,E2 -8081.311} C_VEL
LIN {X 0,Y 460.606,Z 376.608,A -85,B 0,C 180,E1 -8084.059,E2 -8084.059} C_VEL
LIN {X 0,Y 460.633,Z 376.603,A -85,B 0,C 180,E1 -8087.666,E2 -8087.666} C_VEL
LIN {X 0,Y 460.623,Z 376.603,A -85,B 0,C 180,E1 -8091.224,E2 -8091.224} C_VEL
LIN {X 0,Y 460.705,Z 376.596,A -85,B 0,C 180,E1 -8093.87,E2 -8093.87} C_VEL
LIN {X 0,Y 460.803,Z 376.581,A -85,B 0,C 180,E1 -8097.378,E2 -8097.378} C_VEL
LIN {X 0,Y 460.856,Z 376.579,A -85,B 0,C 180,E1 -8100,E2 -8100} C_VEL
LIN {X 0,Y 460.828,Z 376.58,A -85,B 0,C 180,E1 -8102.622,E2 -8102.622} C_VEL
LIN {X 0,Y 460.713,Z 376.6,A -85,B 0,C 180,E1 -8106.13,E2 -8106.13} C_VEL
LIN {X 0,Y 460.63,Z 376.603,A -85,B 0,C 180,E1 -8108.776,E2 -8108.776} C_VEL
LIN {X 0,Y 460.616,Z 376.607,A -85,B 0,C 180,E1 -8112.445,E2 -8112.445} C_VEL
LIN {X 0,Y 460.603,Z 376.614,A -85,B 0,C 180,E1 -8115.998,E2 -8115.998} C_VEL
LIN {X 0,Y 460.574,Z 376.609,A -85,B 0,C 180,E1 -8118.902,E2 -8118.902} C_VEL
LIN {X 0,Y 460.519,Z 376.619,A -85,B 0,C 180,E1 -8121.486,E2 -8121.486} C_VEL
LIN {X 0,Y 460.546,Z 376.615,A -85,B 0,C 180,E1 -8124.332,E2 -8124.332} C_VEL
LIN {X 0,Y 460.582,Z 376.61,A -85,B 0,C 180,E1 -8127.243,E2 -8127.243} C_VEL
LIN {X 0,Y 460.524,Z 376.618,A -85,B 0,C 180,E1 -8130.239,E2 -8130.239} C_VEL
LIN {X 0,Y 460.532,Z 376.618,A -85,B 0,C 180,E1 -8133.325,E2 -8133.325} C_VEL
LIN {X 0,Y 460.481,Z 376.621,A -85,B 0,C 180,E1 -8136.529,E2 -8136.529} C_VEL
LIN {X 0,Y 460.561,Z 376.615,A -85,B 0,C 180,E1 -8139.86,E2 -8139.86} C_VEL
LIN {X 0,Y 460.519,Z 376.617,A -85,B 0,C 180,E1 -8142.901,E2 -8142.901} C_VEL
LIN {X 0,Y 460.514,Z 376.621,A -85,B 0,C 180,E1 -8145.83,E2 -8145.83} C_VEL
LIN {X 0,Y 460.533,Z 376.617,A -85,B 0,C 180,E1 -8148.989,E2 -8148.989} C_VEL
LIN {X 0,Y 460.529,Z 376.621,A -85,B 0,C 180,E1 -8151.267,E2 -8151.267} C_VEL
LIN {X 0,Y 460.517,Z 376.617,A -85,B 0,C 180,E1 -8154.555,E2 -8154.555} C_VEL
LIN {X 0,Y 460.534,Z 376.617,A -85,B 0,C 180,E1 -8157.716,E2 -8157.716} C_VEL
LIN {X 0,Y 460.543,Z 376.615,A -85,B 0,C 180,E1 -8160.769,E2 -8160.769} C_VEL
LIN {X 0,Y 460.566,Z 376.615,A -85,B 0,C 180,E1 -8163.735,E2 -8163.735} C_VEL
LIN {X 0,Y 460.559,Z 376.619,A -85,B 0,C 180,E1 -8167.1,E2 -8167.1} C_VEL
LIN {X 0,Y 460.567,Z 376.728,A -85,B 0,C 180,E1 -8167.456,E2 -8167.456} C_VEL
LIN {X 0,Y 462.147,Z 385.762,A -85,B 0,C 180,E1 -8169.527,E2 -8169.527} C_VEL
LIN {X 0,Y 461.719,Z 396.472,A -85,B 0,C 180,E1 -8171.818,E2 -8171.818} C_VEL
LIN {X 0,Y 461.541,Z 401.053,A -85,B 0,C 180,E1 -8172.782,E2 -8172.782} C_VEL
LIN {X 0,Y 464.531,Z 416.686,A -85,B 0,C 180,E1 -8173.148,E2 -8173.148} C_VEL
LIN {X 0,Y 464.375,Z 443.823,A -85,B 0,C 180,E1 -8173.572,E2 -8173.572} C_VEL
LIN {X 0,Y 463.623,Z 449.669,A -85,B 0,C 180,E1 -8173.637,E2 -8173.637} C_VEL
LIN {X 0,Y 458,Z 468.676,A -85,B 0,C 180,E1 -8173.732,E2 -8173.732} C_VEL
LIN {X 0,Y 457.395,Z 474.516,A -85,B 0,C 180,E1 -8173.804,E2 -8173.804} C_VEL
LIN {X 0,Y 457.053,Z 508.546,A -85,B 0,C 180,E1 -8174.361,E2 -8174.361} C_VEL
LIN {X 0,Y 456.625,Z 521.653,A -85,B 0,C 180,E1 -8174.746,E2 -8174.746} C_VEL
LIN {X 0,Y 456.224,Z 533.714,A -85,B 0,C 180,E1 -8175.275,E2 -8175.275} C_VEL
LIN {X 0,Y 455.763,Z 545.092,A -85,B 0,C 180,E1 -8175.944,E2 -8175.944} C_VEL
LIN {X 0,Y 455.27,Z 556.81,A -85,B 0,C 180,E1 -8176.843,E2 -8176.843} C_VEL
LIN {X 0,Y 454.69,Z 567.232,A -85,B 0,C 180,E1 -8177.843,E2 -8177.843} C_VEL
LIN {X 0,Y 454.17,Z 575.789,A -85,B 0,C 180,E1 -8178.847,E2 -8178.847} C_VEL
LIN {X 0,Y 453.726,Z 583.669,A -85,B 0,C 180,E1 -8179.965,E2 -8179.965} C_VEL
LIN {X 0,Y 453.285,Z 591.373,A -85,B 0,C 180,E1 -8181.305,E2 -8181.305} C_VEL
LIN {X 0,Y 452.887,Z 598.442,A -85,B 0,C 180,E1 -8182.869,E2 -8182.869} C_VEL
LIN {X 0,Y 452.791,Z 603.149,A -85,B 0,C 180,E1 -8184.21,E2 -8184.21} C_VEL
LIN {X 0,Y 452.564,Z 606.757,A -85,B 0,C 180,E1 -8185.547,E2 -8185.547} C_VEL
LIN {X 0,Y 452.583,Z 608.619,A -85,B 0,C 180,E1 -8186.439,E2 -8186.439} C_VEL
LIN {X 0,Y 452.533,Z 610.024,A -85,B 0,C 180,E1 -8187.33,E2 -8187.33} C_VEL
LIN {X 0,Y 452.43,Z 611.639,A -85,B 0,C 180,E1 -8189.11,E2 -8189.11} C_VEL
LIN {X 0,Y 452.408,Z 611.875,A -85,B 0,C 180,E1 -8190,E2 -8190} C_VEL
LIN {X 0,Y 452.43,Z 611.688,A -85,B 0,C 180,E1 -8190.89,E2 -8190.89} C_VEL
LIN {X 0,Y 452.533,Z 610.135,A -85,B 0,C 180,E1 -8192.671,E2 -8192.671} C_VEL
LIN {X 0,Y 452.581,Z 608.779,A -85,B 0,C 180,E1 -8193.561,E2 -8193.561} C_VEL
LIN {X 0,Y 452.593,Z 605.914,A -85,B 0,C 180,E1 -8194.9,E2 -8194.9} C_VEL
LIN {X 0,Y 452.831,Z 602.024,A -85,B 0,C 180,E1 -8196.237,E2 -8196.237} C_VEL
LIN {X 0,Y 452.991,Z 597.01,A -85,B 0,C 180,E1 -8197.578,E2 -8197.578} C_VEL
LIN {X 0,Y 453.332,Z 590.696,A -85,B 0,C 180,E1 -8198.919,E2 -8198.919} C_VEL
LIN {X 0,Y 453.739,Z 582.792,A -85,B 0,C 180,E1 -8200.261,E2 -8200.261} C_VEL
LIN {X 0,Y 454.32,Z 572.959,A -85,B 0,C 180,E1 -8201.602,E2 -8201.602} C_VEL
LIN {X 0,Y 454.913,Z 562.845,A -85,B 0,C 180,E1 -8202.698,E2 -8202.698} C_VEL
LIN {X 0,Y 455.464,Z 551.006,A -85,B 0,C 180,E1 -8203.724,E2 -8203.724} C_VEL
LIN {X 0,Y 456.02,Z 539.417,A -85,B 0,C 180,E1 -8204.504,E2 -8204.504} C_VEL
LIN {X 0,Y 456.512,Z 527.366,A -85,B 0,C 180,E1 -8205.115,E2 -8205.115} C_VEL
LIN {X 0,Y 456.871,Z 514.236,A -85,B 0,C 180,E1 -8205.588,E2 -8205.588} C_VEL
LIN {X 0,Y 457.136,Z 501.562,A -85,B 0,C 180,E1 -8205.865,E2 -8205.865} C_VEL
LIN {X 0,Y 457.738,Z 417.633,A -85,B 0,C 180,E1 -8207.19,E2 -8207.19} C_VEL
LIN {X 0,Y 454.585,Z 401.154,A -85,B 0,C 180,E1 -8207.593,E2 -8207.593} C_VEL
LIN {X 0,Y 455.206,Z 388.469,A -85,B 0,C 180,E1 -8210.328,E2 -8210.328} C_VEL
LIN {X 0,Y 454.804,Z 384.208,A -85,B 0,C 180,E1 -8211.294,E2 -8211.294} C_VEL
LIN {X 0,Y 453.527,Z 377.499,A -85,B 0,C 180,E1 -8212.914,E2 -8212.914} C_VEL
LIN {X 0,Y 453.522,Z 377.496,A -85,B 0,C 180,E1 -8215.999,E2 -8215.999} C_VEL
LIN {X 0,Y 453.514,Z 377.495,A -85,B 0,C 180,E1 -8218.712,E2 -8218.712} C_VEL
LIN {X 0,Y 453.468,Z 377.495,A -85,B 0,C 180,E1 -8221.8,E2 -8221.8} C_VEL
LIN {X 0,Y 453.484,Z 377.497,A -85,B 0,C 180,E1 -8224.989,E2 -8224.989} C_VEL
LIN {X 0,Y 453.467,Z 377.498,A -85,B 0,C 180,E1 -8228.312,E2 -8228.312} C_VEL
LIN {X 0,Y 453.498,Z 377.499,A -85,B 0,C 180,E1 -8230.609,E2 -8230.609} C_VEL
LIN {X 0,Y 453.46,Z 377.497,A -85,B 0,C 180,E1 -8233.244,E2 -8233.244} C_VEL
LIN {X 0,Y 453.478,Z 377.494,A -85,B 0,C 180,E1 -8235.78,E2 -8235.78} C_VEL
LIN {X 0,Y 453.486,Z 377.496,A -85,B 0,C 180,E1 -8238.21,E2 -8238.21} C_VEL
LIN {X 0,Y 453.52,Z 377.492,A -85,B 0,C 180,E1 -8240.79,E2 -8240.79} C_VEL
LIN {X 0,Y 453.459,Z 377.498,A -85,B 0,C 180,E1 -8243.917,E2 -8243.917} C_VEL
LIN {X 0,Y 453.487,Z 377.492,A -85,B 0,C 180,E1 -8247.151,E2 -8247.151} C_VEL
LIN {X 0,Y 453.502,Z 377.498,A -85,B 0,C 180,E1 -8250.27,E2 -8250.27} C_VEL
LIN {X 0,Y 453.509,Z 377.489,A -85,B 0,C 180,E1 -8253.294,E2 -8253.294} C_VEL
LIN {X 0,Y 453.503,Z 377.498,A -85,B 0,C 180,E1 -8256.239,E2 -8256.239} C_VEL
LIN {X 0,Y 453.488,Z 377.492,A -85,B 0,C 180,E1 -8259.118,E2 -8259.118} C_VEL
LIN {X 0,Y 453.518,Z 377.494,A -85,B 0,C 180,E1 -8261.945,E2 -8261.945} C_VEL
LIN {X 0,Y 453.545,Z 377.486,A -85,B 0,C 180,E1 -8264.726,E2 -8264.726} C_VEL
LIN {X 0,Y 453.565,Z 377.486,A -85,B 0,C 180,E1 -8268.379,E2 -8268.379} C_VEL
LIN {X 0,Y 453.657,Z 377.479,A -85,B 0,C 180,E1 -8271.985,E2 -8271.985} C_VEL
LIN {X 0,Y 453.677,Z 377.469,A -85,B 0,C 180,E1 -8274.667,E2 -8274.667} C_VEL
LIN {X 0,Y 453.75,Z 377.461,A -85,B 0,C 180,E1 -8277.337,E2 -8277.337} C_VEL
LIN {X 0,Y 453.829,Z 377.455,A -85,B 0,C 180,E1 -8280,E2 -8280} C_VEL
LIN {X 0,Y 453.75,Z 377.46,A -85,B 0,C 180,E1 -8282.663,E2 -8282.663} C_VEL
LIN {X 0,Y 453.679,Z 377.47,A -85,B 0,C 180,E1 -8286.225,E2 -8286.225} C_VEL
LIN {X 0,Y 453.59,Z 377.48,A -85,B 0,C 180,E1 -8288.913,E2 -8288.913} C_VEL
LIN {X 0,Y 453.607,Z 377.477,A -85,B 0,C 180,E1 -8292.551,E2 -8292.551} C_VEL
LIN {X 0,Y 453.55,Z 377.485,A -85,B 0,C 180,E1 -8296.196,E2 -8296.196} C_VEL
LIN {X 0,Y 453.526,Z 377.49,A -85,B 0,C 180,E1 -8299.041,E2 -8299.041} C_VEL
LIN {X 0,Y 453.481,Z 377.496,A -85,B 0,C 180,E1 -8301.836,E2 -8301.836} C_VEL
LIN {X 0,Y 453.505,Z 377.491,A -85,B 0,C 180,E1 -8304.735,E2 -8304.735} C_VEL
LIN {X 0,Y 453.537,Z 377.487,A -85,B 0,C 180,E1 -8307.959,E2 -8307.959} C_VEL
LIN {X 0,Y 453.47,Z 377.5,A -85,B 0,C 180,E1 -8311.525,E2 -8311.525} C_VEL
LIN {X 0,Y 453.486,Z 377.494,A -85,B 0,C 180,E1 -8314.776,E2 -8314.776} C_VEL
LIN {X 0,Y 453.467,Z 377.495,A -85,B 0,C 180,E1 -8318.312,E2 -8318.312} C_VEL
LIN {X 0,Y 453.497,Z 377.492,A -85,B 0,C 180,E1 -8320.609,E2 -8320.609} C_VEL
LIN {X 0,Y 453.476,Z 377.494,A -85,B 0,C 180,E1 -8324.22,E2 -8324.22} C_VEL
LIN {X 0,Y 453.468,Z 377.502,A -85,B 0,C 180,E1 -8327.005,E2 -8327.005} C_VEL
LIN {X 0,Y 453.509,Z 377.492,A -85,B 0,C 180,E1 -8330.552,E2 -8330.552} C_VEL
LIN {X 0,Y 453.458,Z 377.496,A -85,B 0,C 180,E1 -8333.917,E2 -8333.917} C_VEL
LIN {X 0,Y 453.486,Z 377.497,A -85,B 0,C 180,E1 -8337.151,E2 -8337.151} C_VEL
LIN {X 0,Y 453.479,Z 377.498,A -85,B 0,C 180,E1 -8340.268,E2 -8340.268} C_VEL
LIN {X 0,Y 453.51,Z 377.496,A -85,B 0,C 180,E1 -8343.294,E2 -8343.294} C_VEL
LIN {X 0,Y 453.547,Z 377.604,A -85,B 0,C 180,E1 -8344.092,E2 -8344.092} C_VEL
LIN {X 0,Y 455.907,Z 389.848,A -85,B 0,C 180,E1 -8346.612,E2 -8346.612} C_VEL
LIN {X 0,Y 455.318,Z 402.298,A -85,B 0,C 180,E1 -8348.969,E2 -8348.969} C_VEL
LIN {X 0,Y 454.547,Z 418.415,A -85,B 0,C 180,E1 -8351.987,E2 -8351.987} C_VEL
LIN {X 0,Y 454.429,Z 420.857,A -85,B 0,C 180,E1 -8352.443,E2 -8352.443} C_VEL
LIN {X 0,Y 457.678,Z 441.765,A -85,B 0,C 180,E1 -8352.91,E2 -8352.91} C_VEL
LIN {X 0,Y 456.937,Z 528.86,A -85,B 0,C 180,E1 -8354.3,E2 -8354.3} C_VEL
LIN {X 0,Y 456.516,Z 542.128,A -85,B 0,C 180,E1 -8354.685,E2 -8354.685} C_VEL
LIN {X 0,Y 456.033,Z 554.289,A -85,B 0,C 180,E1 -8355.212,E2 -8355.212} C_VEL
LIN {X 0,Y 455.481,Z 566.558,A -85,B 0,C 180,E1 -8355.935,E2 -8355.935} C_VEL
LIN {X 0,Y 454.839,Z 577.509,A -85,B 0,C 180,E1 -8356.769,E2 -8356.769} C_VEL
LIN {X 0,Y 454.371,Z 588.593,A -85,B 0,C 180,E1 -8357.834,E2 -8357.834} C_VEL
LIN {X 0,Y 453.861,Z 597.127,A -85,B 0,C 180,E1 -8358.839,E2 -8358.839} C_VEL
LIN {X 0,Y 453.43,Z 605.002,A -85,B 0,C 180,E1 -8359.958,E2 -8359.958} C_VEL
LIN {X 0,Y 453.017,Z 612.693,A -85,B 0,C 180,E1 -8361.3,E2 -8361.3} C_VEL
LIN {X 0,Y 452.724,Z 619.784,A -85,B 0,C 180,E1 -8362.866,E2 -8362.866} C_VEL
LIN {X 0,Y 452.585,Z 624.502,A -85,B 0,C 180,E1 -8364.207,E2 -8364.207} C_VEL
LIN {X 0,Y 452.488,Z 628.107,A -85,B 0,C 180,E1 -8365.546,E2 -8365.546} C_VEL
LIN {X 0,Y 452.456,Z 629.966,A -85,B 0,C 180,E1 -8366.438,E2 -8366.438} C_VEL
LIN {X 0,Y 452.503,Z 631.362,A -85,B 0,C 180,E1 -8367.329,E2 -8367.329} C_VEL
LIN {X 0,Y 452.403,Z 632.962,A -85,B 0,C 180,E1 -8369.11,E2 -8369.11} C_VEL
LIN {X 0,Y 452.406,Z 633.179,A -85,B 0,C 180,E1 -8370,E2 -8370} C_VEL
LIN {X 0,Y 452.436,Z 632.357,A -85,B 0,C 180,E1 -8371.78,E2 -8371.78} C_VEL
LIN {X 0,Y 452.503,Z 631.364,A -85,B 0,C 180,E1 -8372.67,E2 -8372.67} C_VEL
LIN {X 0,Y 452.455,Z 629.968,A -85,B 0,C 180,E1 -8373.562,E2 -8373.562} C_VEL
LIN {X 0,Y 452.554,Z 627.036,A -85,B 0,C 180,E1 -8374.9,E2 -8374.9} C_VEL
LIN {X 0,Y 452.628,Z 622.456,A -85,B 0,C 180,E1 -8376.416,E2 -8376.416} C_VEL
LIN {X 0,Y 452.891,Z 615.95,A -85,B 0,C 180,E1 -8378.028,E2 -8378.028} C_VEL
LIN {X 0,Y 453.201,Z 609.053,A -85,B 0,C 180,E1 -8379.371,E2 -8379.371} C_VEL
LIN {X 0,Y 453.628,Z 600.426,A -85,B 0,C 180,E1 -8380.714,E2 -8380.714} C_VEL
LIN {X 0,Y 454.205,Z 591.581,A -85,B 0,C 180,E1 -8381.831,E2 -8381.831} C_VEL
LIN {X 0,Y 454.714,Z 581.107,A -85,B 0,C 180,E1 -8382.91,E2 -8382.91} C_VEL
LIN {X 0,Y 455.209,Z 571.244,A -85,B 0,C 180,E1 -8383.732,E2 -8383.732} C_VEL
LIN {X 0,Y 455.748,Z 559.378,A -85,B 0,C 180,E1 -8384.512,E2 -8384.512} C_VEL
LIN {X 0,Y 456.349,Z 547.033,A -85,B 0,C 180,E1 -8385.12,E2 -8385.12} C_VEL
LIN {X 0,Y 456.745,Z 534.36,A -85,B 0,C 180,E1 -8385.564,E2 -8385.564} C_VEL
LIN {X 0,Y 457.063,Z 521.113,A -85,B 0,C 180,E1 -8385.839,E2 -8385.839} C_VEL
LIN {X 0,Y 457.561,Z 440.237,A -85,B 0,C 180,E1 -8387.117,E2 -8387.117} C_VEL
LIN {X 0,Y 454.419,Z 420.822,A -85,B 0,C 180,E1 -8387.559,E2 -8387.559} C_VEL
LIN {X 0,Y 455.181,Z 406.008,A -85,B 0,C 180,E1 -8390.328,E2 -8390.328} C_VEL
LIN {X 0,Y 455.966,Z 391.08,A -85,B 0,C 180,E1 -8393.144,E2 -8393.144} C_VEL
LIN {X 0,Y 454.538,Z 382.317,A -85,B 0,C 180,E1 -8394.919,E2 -8394.919} C_VEL
LIN {X 0,Y 453.539,Z 377.49,A -85,B 0,C 180,E1 -8395.953,E2 -8395.953} C_VEL
LIN {X 0,Y 453.514,Z 377.495,A -85,B 0,C 180,E1 -8398.712,E2 -8398.712} C_VEL
LIN {X 0,Y 453.467,Z 377.495,A -85,B 0,C 180,E1 -8401.799,E2 -8401.799} C_VEL
LIN {X 0,Y 453.482,Z 377.5,A -85,B 0,C 180,E1 -8404.989,E2 -8404.989} C_VEL
LIN {X 0,Y 453.467,Z 377.495,A -85,B 0,C 180,E1 -8408.311,E2 -8408.311} C_VEL
LIN {X 0,Y 453.496,Z 377.494,A -85,B 0,C 180,E1 -8410.609,E2 -8410.609} C_VEL
LIN {X 0,Y 453.458,Z 377.5,A -85,B 0,C 180,E1 -8413.244,E2 -8413.244} C_VEL
LIN {X 0,Y 453.475,Z 377.494,A -85,B 0,C 180,E1 -8415.78,E2 -8415.78} C_VEL
LIN {X 0,Y 453.484,Z 377.494,A -85,B 0,C 180,E1 -8418.21,E2 -8418.21} C_VEL
LIN {X 0,Y 453.512,Z 377.497,A -85,B 0,C 180,E1 -8420.791,E2 -8420.791} C_VEL
LIN {X 0,Y 453.456,Z 377.496,A -85,B 0,C 180,E1 -8423.917,E2 -8423.917} C_VEL
LIN {X 0,Y 453.485,Z 377.495,A -85,B 0,C 180,E1 -8427.151,E2 -8427.151} C_VEL
LIN {X 0,Y 453.477,Z 377.496,A -85,B 0,C 180,E1 -8430.268,E2 -8430.268} C_VEL
LIN {X 0,Y 453.507,Z 377.491,A -85,B 0,C 180,E1 -8433.294,E2 -8433.294} C_VEL
LIN {X 0,Y 453.5,Z 377.494,A -85,B 0,C 180,E1 -8436.239,E2 -8436.239} C_VEL
LIN {X 0,Y 453.485,Z 377.494,A -85,B 0,C 180,E1 -8439.118,E2 -8439.118} C_VEL
LIN {X 0,Y 453.513,Z 377.491,A -85,B 0,C 180,E1 -8441.945,E2 -8441.945} C_VEL
LIN {X 0,Y 453.542,Z 377.49,A -85,B 0,C 180,E1 -8444.726,E2 -8444.726} C_VEL
LIN {X 0,Y 453.605,Z 377.477,A -85,B 0,C 180,E1 -8447.472,E2 -8447.472} C_VEL
LIN {X 0,Y 453.589,Z 377.48,A -85,B 0,C 180,E1 -8451.087,E2 -8451.087} C_VEL
LIN {X 0,Y 453.672,Z 377.471,A -85,B 0,C 180,E1 -8453.775,E2 -8453.775} C_VEL
LIN {X 0,Y 453.747,Z 377.46,A -85,B 0,C 180,E1 -8457.337,E2 -8457.337} C_VEL
LIN {X 0,Y 453.826,Z 377.455,A -85,B 0,C 180,E1 -8460,E2 -8460} C_VEL
LIN {X 0,Y 453.768,Z 377.459,A -85,B 0,C 180,E1 -8462.663,E2 -8462.663} C_VEL
LIN {X 0,Y 453.681,Z 377.475,A -85,B 0,C 180,E1 -8466.225,E2 -8466.225} C_VEL
LIN {X 0,Y 453.594,Z 377.479,A -85,B 0,C 180,E1 -8468.913,E2 -8468.913} C_VEL
LIN {X 0,Y 453.566,Z 377.484,A -85,B 0,C 180,E1 -8472.529,E2 -8472.529} C_VEL
LIN {X 0,Y 453.548,Z 377.489,A -85,B 0,C 180,E1 -8476.196,E2 -8476.196} C_VEL
LIN {X 0,Y 453.524,Z 377.488,A -85,B 0,C 180,E1 -8479.041,E2 -8479.041} C_VEL
LIN {X 0,Y 453.48,Z 377.501,A -85,B 0,C 180,E1 -8481.836,E2 -8481.836} C_VEL
LIN {X 0,Y 453.517,Z 377.488,A -85,B 0,C 180,E1 -8484.734,E2 -8484.734} C_VEL
LIN {X 0,Y 453.54,Z 377.491,A -85,B 0,C 180,E1 -8487.961,E2 -8487.961} C_VEL
LIN {X 0,Y 453.484,Z 377.493,A -85,B 0,C 180,E1 -8490.759,E2 -8490.759} C_VEL
LIN {X 0,Y 453.48,Z 377.498,A -85,B 0,C 180,E1 -8493.913,E2 -8493.913} C_VEL
LIN {X 0,Y 453.473,Z 377.496,A -85,B 0,C 180,E1 -8497.188,E2 -8497.188} C_VEL
LIN {X 0,Y 453.519,Z 377.494,A -85,B 0,C 180,E1 -8499.447,E2 -8499.447} C_VEL
LIN {X 0,Y 453.471,Z 377.496,A -85,B 0,C 180,E1 -8502.994,E2 -8502.994} C_VEL
LIN {X 0,Y 453.469,Z 377.499,A -85,B 0,C 180,E1 -8505.779,E2 -8505.779} C_VEL
LIN {X 0,Y 453.481,Z 377.493,A -85,B 0,C 180,E1 -8508.209,E2 -8508.209} C_VEL
LIN {X 0,Y 453.497,Z 377.492,A -85,B 0,C 180,E1 -8510.793,E2 -8510.793} C_VEL
LIN {X 0,Y 453.46,Z 377.497,A -85,B 0,C 180,E1 -8513.918,E2 -8513.918} C_VEL
LIN {X 0,Y 453.486,Z 377.498,A -85,B 0,C 180,E1 -8517.151,E2 -8517.151} C_VEL
LIN {X 0,Y 453.478,Z 377.493,A -85,B 0,C 180,E1 -8520.268,E2 -8520.268} C_VEL
LIN {X 0,Y 453.51,Z 377.497,A -85,B 0,C 180,E1 -8523.294,E2 -8523.294} C_VEL
LIN {X 0,Y 453.506,Z 377.496,A -85,B 0,C 180,E1 -8526.239,E2 -8526.239} C_VEL
LIN {X 0,Y 453.532,Z 377.673,A -85,B 0,C 180,E1 -8527.267,E2 -8527.267} C_VEL
LIN {X 0,Y 455.194,Z 386.978,A -85,B 0,C 180,E1 -8529.436,E2 -8529.436} C_VEL
LIN {X 0,Y 454.73,Z 397.713,A -85,B 0,C 180,E1 -8531.762,E2 -8531.762} C_VEL
LIN {X 0,Y 454.588,Z 401.22,A -85,B 0,C 180,E1 -8532.51,E2 -8532.51} C_VEL
LIN {X 0,Y 457.834,Z 418.955,A -85,B 0,C 180,E1 -8532.928,E2 -8532.928} C_VEL
LIN {X 0,Y 457.395,Z 474.516,A -85,B 0,C 180,E1 -8533.804,E2 -8533.804} C_VEL
LIN {X 0,Y 456.738,Z 480.371,A -85,B 0,C 180,E1 -8533.871,E2 -8533.871} C_VEL
LIN {X 0,Y 450.864,Z 499.356,A -85,B 0,C 180,E1 -8533.959,E2 -8533.959} C_VEL
LIN {X 0,Y 450.234,Z 505.192,A -85,B 0,C 180,E1 -8534.044,E2 -8534.044} C_VEL
LIN {X 0,Y 449.926,Z 518.757,A -85,B 0,C 180,E1 -8534.398,E2 -8534.398} C_VEL
LIN {X 0,Y 449.447,Z 531.634,A -85,B 0,C 180,E1 -8534.932,E2 -8534.932} C_VEL
LIN {X 0,Y 448.953,Z 543.519,A -85,B 0,C 180,E1 -8535.611,E2 -8535.611} C_VEL
LIN {X 0,Y 448.481,Z 554.29,A -85,B 0,C 180,E1 -8536.405,E2 -8536.405} C_VEL
LIN {X 0,Y 447.899,Z 565.271,A -85,B 0,C 180,E1 -8537.425,E2 -8537.425} C_VEL
LIN {X 0,Y 447.305,Z 574.184,A -85,B 0,C 180,E1 -8538.444,E2 -8538.444} C_VEL
LIN {X 0,Y 446.713,Z 583.839,A -85,B 0,C 180,E1 -8539.805,E2 -8539.805} C_VEL
LIN {X 0,Y 446.249,Z 591.543,A -85,B 0,C 180,E1 -8541.167,E2 -8541.167} C_VEL
LIN {X 0,Y 445.841,Z 598.611,A -85,B 0,C 180,E1 -8542.755,E2 -8542.755} C_VEL
LIN {X 0,Y 445.721,Z 603.318,A -85,B 0,C 180,E1 -8544.118,E2 -8544.118} C_VEL
LIN {X 0,Y 445.484,Z 606.925,A -85,B 0,C 180,E1 -8545.476,E2 -8545.476} C_VEL
LIN {X 0,Y 445.485,Z 608.787,A -85,B 0,C 180,E1 -8546.382,E2 -8546.382} C_VEL
LIN {X 0,Y 445.461,Z 610.191,A -85,B 0,C 180,E1 -8547.287,E2 -8547.287} C_VEL
LIN {X 0,Y 445.341,Z 611.806,A -85,B 0,C 180,E1 -8549.096,E2 -8549.096} C_VEL
LIN {X 0,Y 445.317,Z 612.042,A -85,B 0,C 180,E1 -8550,E2 -8550} C_VEL
LIN {X 0,Y 445.341,Z 611.854,A -85,B 0,C 180,E1 -8550.904,E2 -8550.904} C_VEL
LIN {X 0,Y 445.461,Z 610.301,A -85,B 0,C 180,E1 -8552.713,E2 -8552.713} C_VEL
LIN {X 0,Y 445.483,Z 608.945,A -85,B 0,C 180,E1 -8553.618,E2 -8553.618} C_VEL
LIN {X 0,Y 445.532,Z 606.08,A -85,B 0,C 180,E1 -8554.977,E2 -8554.977} C_VEL
LIN {X 0,Y 445.766,Z 602.19,A -85,B 0,C 180,E1 -8556.336,E2 -8556.336} C_VEL
LIN {X 0,Y 445.958,Z 597.175,A -85,B 0,C 180,E1 -8557.698,E2 -8557.698} C_VEL
LIN {X 0,Y 446.298,Z 590.861,A -85,B 0,C 180,E1 -8559.06,E2 -8559.06} C_VEL
LIN {X 0,Y 446.762,Z 582.956,A -85,B 0,C 180,E1 -8560.423,E2 -8560.423} C_VEL
LIN {X 0,Y 447.36,Z 573.122,A -85,B 0,C 180,E1 -8561.785,E2 -8561.785} C_VEL
LIN {X 0,Y 447.98,Z 563.142,A -85,B 0,C 180,E1 -8562.885,E2 -8562.885} C_VEL
LIN {X 0,Y 448.501,Z 552.59,A -85,B 0,C 180,E1 -8563.825,E2 -8563.825} C_VEL
LIN {X 0,Y 449.076,Z 541.402,A -85,B 0,C 180,E1 -8564.617,E2 -8564.617} C_VEL
LIN {X 0,Y 449.58,Z 530.059,A -85,B 0,C 180,E1 -8565.238,E2 -8565.238} C_VEL
LIN {X 0,Y 449.979,Z 517.133,A -85,B 0,C 180,E1 -8565.746,E2 -8565.746} C_VEL
LIN {X 0,Y 450.267,Z 503.319,A -85,B 0,C 180,E1 -8566.085,E2 -8566.085} C_VEL
LIN {X 0,Y 450.939,Z 418.266,A -85,B 0,C 180,E1 -8567.449,E2 -8567.449} C_VEL
LIN {X 0,Y 447.652,Z 401.314,A -85,B 0,C 180,E1 -8567.875,E2 -8567.875} C_VEL
LIN {X 0,Y 448.301,Z 388.614,A -85,B 0,C 180,E1 -8570.655,E2 -8570.655} C_VEL
LIN {X 0,Y 446.497,Z 378.375,A -85,B 0,C 180,E1 -8573.112,E2 -8573.112} C_VEL
LIN {X 0,Y 446.479,Z 378.372,A -85,B 0,C 180,E1 -8576.203,E2 -8576.203} C_VEL
LIN {X 0,Y 446.453,Z 378.371,A -85,B 0,C 180,E1 -8579.209,E2 -8579.209} C_VEL
LIN {X 0,Y 446.426,Z 378.375,A -85,B 0,C 180,E1 -8582.362,E2 -8582.362} C_VEL
LIN {X 0,Y 446.423,Z 378.372,A -85,B 0,C 180,E1 -8585.626,E2 -8585.626} C_VEL
LIN {X 0,Y 446.445,Z 378.373,A -85,B 0,C 180,E1 -8589.027,E2 -8589.027} C_VEL
LIN {X 0,Y 446.438,Z 378.374,A -85,B 0,C 180,E1 -8592.277,E2 -8592.277} C_VEL
LIN {X 0,Y 446.46,Z 378.369,A -85,B 0,C 180,E1 -8595.103,E2 -8595.103} C_VEL
LIN {X 0,Y 446.434,Z 378.377,A -85,B 0,C 180,E1 -8598.609,E2 -8598.609} C_VEL
LIN {X 0,Y 446.465,Z 378.369,A -85,B 0,C 180,E1 -8600.975,E2 -8600.975} C_VEL
LIN {X 0,Y 446.423,Z 378.38,A -85,B 0,C 180,E1 -8604.374,E2 -8604.374} C_VEL
LIN {X 0,Y 446.427,Z 378.372,A -85,B 0,C 180,E1 -8607.639,E2 -8607.639} C_VEL
LIN {X 0,Y 446.464,Z 378.369,A -85,B 0,C 180,E1 -8610.792,E2 -8610.792} C_VEL
LIN {X 0,Y 446.483,Z 378.368,A -85,B 0,C 180,E1 -8613.849,E2 -8613.849} C_VEL
LIN {X 0,Y 446.431,Z 378.372,A -85,B 0,C 180,E1 -8616.823,E2 -8616.823} C_VEL
LIN {X 0,Y 446.45,Z 378.371,A -85,B 0,C 180,E1 -8619.737,E2 -8619.737} C_VEL
LIN {X 0,Y 446.469,Z 378.369,A -85,B 0,C 180,E1 -8622.597,E2 -8622.597} C_VEL
LIN {X 0,Y 446.476,Z 378.367,A -85,B 0,C 180,E1 -8625.412,E2 -8625.412} C_VEL
LIN {X 0,Y 446.523,Z 378.365,A -85,B 0,C 180,E1 -8628.193,E2 -8628.193} C_VEL
LIN {X 0,Y 446.606,Z 378.356,A -85,B 0,C 180,E1 -8631.858,E2 -8631.858} C_VEL
LIN {X 0,Y 446.651,Z 378.345,A -85,B 0,C 180,E1 -8634.583,E2 -8634.583} C_VEL
LIN {X 0,Y 446.67,Z 378.345,A -85,B 0,C 180,E1 -8638.197,E2 -8638.197} C_VEL
LIN {X 0,Y 446.798,Z 378.331,A -85,B 0,C 180,E1 -8640,E2 -8640} C_VEL
LIN {X 0,Y 446.697,Z 378.338,A -85,B 0,C 180,E1 -8642.705,E2 -8642.705} C_VEL
LIN {X 0,Y 446.646,Z 378.346,A -85,B 0,C 180,E1 -8646.324,E2 -8646.324} C_VEL
LIN {X 0,Y 446.538,Z 378.359,A -85,B 0,C 180,E1 -8649.055,E2 -8649.055} C_VEL
LIN {X 0,Y 446.539,Z 378.358,A -85,B 0,C 180,E1 -8652.729,E2 -8652.729} C_VEL
LIN {X 0,Y 446.495,Z 378.363,A -85,B 0,C 180,E1 -8656.459,E2 -8656.459} C_VEL
LIN {X 0,Y 446.475,Z 378.371,A -85,B 0,C 180,E1 -8659.303,E2 -8659.303} C_VEL
LIN {X 0,Y 446.422,Z 378.373,A -85,B 0,C 180,E1 -8662.199,E2 -8662.199} C_VEL
LIN {X 0,Y 446.449,Z 378.373,A -85,B 0,C 180,E1 -8665.153,E2 -8665.153} C_VEL
LIN {X 0,Y 446.489,Z 378.364,A -85,B 0,C 180,E1 -8668.178,E2 -8668.178} C_VEL
LIN {X 0,Y 446.423,Z 378.375,A -85,B 0,C 180,E1 -8671.775,E2 -8671.775} C_VEL
LIN {X 0,Y 446.427,Z 378.372,A -85,B 0,C 180,E1 -8674.523,E2 -8674.523} C_VEL
LIN {X 0,Y 446.418,Z 378.373,A -85,B 0,C 180,E1 -8678.079,E2 -8678.079} C_VEL
LIN {X 0,Y 446.431,Z 378.376,A -85,B 0,C 180,E1 -8680.917,E2 -8680.917} C_VEL
LIN {X 0,Y 446.426,Z 378.372,A -85,B 0,C 180,E1 -8683.843,E2 -8683.843} C_VEL
LIN {X 0,Y 446.403,Z 378.375,A -85,B 0,C 180,E1 -8686.403,E2 -8686.403} C_VEL
LIN {X 0,Y 446.431,Z 378.379,A -85,B 0,C 180,E1 -8689.082,E2 -8689.082} C_VEL
LIN {X 0,Y 446.419,Z 378.373,A -85,B 0,C 180,E1 -8691.92,E2 -8691.92} C_VEL
LIN {X 0,Y 446.433,Z 378.373,A -85,B 0,C 180,E1 -8695.477,E2 -8695.477} C_VEL
LIN {X 0,Y 446.42,Z 378.378,A -85,B 0,C 180,E1 -8698.7,E2 -8698.7} C_VEL
LIN {X 0,Y 446.488,Z 378.369,A -85,B 0,C 180,E1 -8701.821,E2 -8701.821} C_VEL
LIN {X 0,Y 446.481,Z 378.439,A -85,B 0,C 180,E1 -8703.848,E2 -8703.848} C_VEL
LIN {X 0,Y 448.708,Z 389.698,A -85,B 0,C 180,E1 -8706.214,E2 -8706.214} C_VEL
LIN {X 0,Y 448.919,Z 393.438,A -85,B 0,C 180,E1 -8706.959,E2 -8706.959} C_VEL
LIN {X 0,Y 447.99,Z 410.721,A -85,B 0,C 180,E1 -8710.266,E2 -8710.266} C_VEL
LIN {X 0,Y 447.474,Z 420.683,A -85,B 0,C 180,E1 -8712.159,E2 -8712.159} C_VEL
LIN {X 0,Y 450.893,Z 441.615,A -85,B 0,C 180,E1 -8712.644,E2 -8712.644} C_VEL
LIN {X 0,Y 450.104,Z 528.704,A -85,B 0,C 180,E1 -8714.055,E2 -8714.055} C_VEL
LIN {X 0,Y 449.68,Z 541.969,A -85,B 0,C 180,E1 -8714.447,E2 -8714.447} C_VEL
LIN {X 0,Y 449.151,Z 554.126,A -85,B 0,C 180,E1 -8714.98,E2 -8714.98} C_VEL
LIN {X 0,Y 448.574,Z 566.394,A -85,B 0,C 180,E1 -8715.714,E2 -8715.714} C_VEL
LIN {X 0,Y 447.847,Z 578.318,A -85,B 0,C 180,E1 -8716.646,E2 -8716.646} C_VEL
LIN {X 0,Y 447.35,Z 589.472,A -85,B 0,C 180,E1 -8717.755,E2 -8717.755} C_VEL
LIN {X 0,Y 446.761,Z 598.639,A -85,B 0,C 180,E1 -8718.889,E2 -8718.889} C_VEL
LIN {X 0,Y 446.222,Z 607.572,A -85,B 0,C 180,E1 -8720.252,E2 -8720.252} C_VEL
LIN {X 0,Y 445.861,Z 614.764,A -85,B 0,C 180,E1 -8721.616,E2 -8721.616} C_VEL
LIN {X 0,Y 445.669,Z 619.618,A -85,B 0,C 180,E1 -8722.752,E2 -8722.752} C_VEL
LIN {X 0,Y 445.496,Z 623.737,A -85,B 0,C 180,E1 -8723.924,E2 -8723.924} C_VEL
LIN {X 0,Y 445.414,Z 627.94,A -85,B 0,C 180,E1 -8725.475,E2 -8725.475} C_VEL
LIN {X 0,Y 445.355,Z 629.799,A -85,B 0,C 180,E1 -8726.381,E2 -8726.381} C_VEL
LIN {X 0,Y 445.427,Z 631.195,A -85,B 0,C 180,E1 -8727.287,E2 -8727.287} C_VEL
LIN {X 0,Y 445.315,Z 632.796,A -85,B 0,C 180,E1 -8729.096,E2 -8729.096} C_VEL
LIN {X 0,Y 445.316,Z 633.012,A -85,B 0,C 180,E1 -8730,E2 -8730} C_VEL
LIN {X 0,Y 445.355,Z 632.189,A -85,B 0,C 180,E1 -8731.808,E2 -8731.808} C_VEL
LIN {X 0,Y 445.427,Z 631.197,A -85,B 0,C 180,E1 -8732.713,E2 -8732.713} C_VEL
LIN {X 0,Y 445.355,Z 629.8,A -85,B 0,C 180,E1 -8733.619,E2 -8733.619} C_VEL
LIN {X 0,Y 445.485,Z 626.869,A -85,B 0,C 180,E1 -8734.978,E2 -8734.978} C_VEL
LIN {X 0,Y 445.575,Z 621.467,A -85,B 0,C 180,E1 -8736.748,E2 -8736.748} C_VEL
LIN {X 0,Y 445.844,Z 615.781,A -85,B 0,C 180,E1 -8738.156,E2 -8738.156} C_VEL
LIN {X 0,Y 446.151,Z 608.884,A -85,B 0,C 180,E1 -8739.52,E2 -8739.52} C_VEL
LIN {X 0,Y 446.631,Z 600.256,A -85,B 0,C 180,E1 -8740.884,E2 -8740.884} C_VEL
LIN {X 0,Y 447.206,Z 591.41,A -85,B 0,C 180,E1 -8742.018,E2 -8742.018} C_VEL
LIN {X 0,Y 447.813,Z 580.594,A -85,B 0,C 180,E1 -8743.146,E2 -8743.146} C_VEL
LIN {X 0,Y 448.385,Z 569.533,A -85,B 0,C 180,E1 -8744.06,E2 -8744.06} C_VEL
LIN {X 0,Y 449.003,Z 557.215,A -85,B 0,C 180,E1 -8744.851,E2 -8744.851} C_VEL
LIN {X 0,Y 449.562,Z 545.558,A -85,B 0,C 180,E1 -8745.412,E2 -8745.412} C_VEL
LIN {X 0,Y 449.942,Z 533.159,A -85,B 0,C 180,E1 -8745.834,E2 -8745.834} C_VEL
LIN {X 0,Y 450.27,Z 517.349,A -85,B 0,C 180,E1 -8746.142,E2 -8746.142} C_VEL
LIN {X 0,Y 450.729,Z 440.748,A -85,B 0,C 180,E1 -8747.373,E2 -8747.373} C_VEL
LIN {X 0,Y 447.452,Z 420.698,A -85,B 0,C 180,E1 -8747.833,E2 -8747.833} C_VEL
LIN {X 0,Y 448.223,Z 405.85,A -85,B 0,C 180,E1 -8750.658,E2 -8750.658} C_VEL
LIN {X 0,Y 449.027,Z 392.177,A -85,B 0,C 180,E1 -8753.279,E2 -8753.279} C_VEL
LIN {X 0,Y 447.263,Z 382.166,A -85,B 0,C 180,E1 -8755.353,E2 -8755.353} C_VEL
LIN {X 0,Y 446.477,Z 378.369,A -85,B 0,C 180,E1 -8756.202,E2 -8756.202} C_VEL
LIN {X 0,Y 446.452,Z 378.376,A -85,B 0,C 180,E1 -8759.209,E2 -8759.209} C_VEL
LIN {X 0,Y 446.425,Z 378.372,A -85,B 0,C 180,E1 -8762.361,E2 -8762.361} C_VEL
LIN {X 0,Y 446.421,Z 378.374,A -85,B 0,C 180,E1 -8765.626,E2 -8765.626} C_VEL
LIN {X 0,Y 446.458,Z 378.376,A -85,B 0,C 180,E1 -8769.026,E2 -8769.026} C_VEL
LIN {X 0,Y 446.436,Z 378.371,A -85,B 0,C 180,E1 -8772.277,E2 -8772.277} C_VEL
LIN {X 0,Y 446.458,Z 378.373,A -85,B 0,C 180,E1 -8775.103,E2 -8775.103} C_VEL
LIN {X 0,Y 446.432,Z 378.376,A -85,B 0,C 180,E1 -8778.609,E2 -8778.609} C_VEL
LIN {X 0,Y 446.457,Z 378.374,A -85,B 0,C 180,E1 -8780.974,E2 -8780.974} C_VEL
LIN {X 0,Y 446.421,Z 378.375,A -85,B 0,C 180,E1 -8784.374,E2 -8784.374} C_VEL
LIN {X 0,Y 446.424,Z 378.372,A -85,B 0,C 180,E1 -8787.639,E2 -8787.639} C_VEL
LIN {X 0,Y 446.452,Z 378.375,A -85,B 0,C 180,E1 -8790.791,E2 -8790.791} C_VEL
LIN {X 0,Y 446.48,Z 378.365,A -85,B 0,C 180,E1 -8793.848,E2 -8793.848} C_VEL
LIN {X 0,Y 446.429,Z 378.376,A -85,B 0,C 180,E1 -8796.823,E2 -8796.823} C_VEL
LIN {X 0,Y 446.447,Z 378.369,A -85,B 0,C 180,E1 -8799.737,E2 -8799.737} C_VEL
LIN {X 0,Y 446.465,Z 378.373,A -85,B 0,C 180,E1 -8802.597,E2 -8802.597} C_VEL
LIN {X 0,Y 446.473,Z 378.366,A -85,B 0,C 180,E1 -8805.412,E2 -8805.412} C_VEL
LIN {X 0,Y 446.542,Z 378.362,A -85,B 0,C 180,E1 -8808.194,E2 -8808.194} C_VEL
LIN {X 0,Y 446.537,Z 378.359,A -85,B 0,C 180,E1 -8810.945,E2 -8810.945} C_VEL
LIN {X 0,Y 446.64,Z 378.346,A -85,B 0,C 180,E1 -8813.676,E2 -8813.676} C_VEL
LIN {X 0,Y 446.694,Z 378.338,A -85,B 0,C 180,E1 -8817.295,E2 -8817.295} C_VEL
LIN {X 0,Y 446.796,Z 378.331,A -85,B 0,C 180,E1 -8820,E2 -8820} C_VEL
LIN {X 0,Y 446.712,Z 378.338,A -85,B 0,C 180,E1 -8822.705,E2 -8822.705} C_VEL
LIN {X 0,Y 446.65,Z 378.349,A -85,B 0,C 180,E1 -8826.324,E2 -8826.324} C_VEL
LIN {X 0,Y 446.54,Z 378.358,A -85,B 0,C 180,E1 -8829.055,E2 -8829.055} C_VEL
LIN {X 0,Y 446.524,Z 378.36,A -85,B 0,C 180,E1 -8832.73,E2 -8832.73} C_VEL
LIN {X 0,Y 446.499,Z 378.367,A -85,B 0,C 180,E1 -8836.228,E2 -8836.228} C_VEL
LIN {X 0,Y 446.473,Z 378.367,A -85,B 0,C 180,E1 -8839.303,E2 -8839.303} C_VEL
LIN {X 0,Y 446.422,Z 378.376,A -85,B 0,C 180,E1 -8842.2,E2 -8842.2} C_VEL
LIN {X 0,Y 446.461,Z 378.368,A -85,B 0,C 180,E1 -8845.152,E2 -8845.152} C_VEL
LIN {X 0,Y 446.487,Z 378.367,A -85,B 0,C 180,E1 -8848.179,E2 -8848.179} C_VEL
LIN {X 0,Y 446.42,Z 378.375,A -85,B 0,C 180,E1 -8851.3,E2 -8851.3} C_VEL
LIN {X 0,Y 446.433,Z 378.371,A -85,B 0,C 180,E1 -8854.523,E2 -8854.523} C_VEL
LIN {X 0,Y 446.433,Z 378.373,A -85,B 0,C 180,E1 -8858.082,E2 -8858.082} C_VEL
LIN {X 0,Y 446.43,Z 378.372,A -85,B 0,C 180,E1 -8860.918,E2 -8860.918} C_VEL
LIN {X 0,Y 446.425,Z 378.376,A -85,B 0,C 180,E1 -8863.843,E2 -8863.843} C_VEL
LIN {X 0,Y 446.402,Z 378.375,A -85,B 0,C 180,E1 -8866.403,E2 -8866.403} C_VEL
LIN {X 0,Y 446.429,Z 378.375,A -85,B 0,C 180,E1 -8869.083,E2 -8869.083} C_VEL
LIN {X 0,Y 446.431,Z 378.372,A -85,B 0,C 180,E1 -8872.123,E2 -8872.123} C_VEL
LIN {X 0,Y 446.434,Z 378.377,A -85,B 0,C 180,E1 -8875.477,E2 -8875.477} C_VEL
LIN {X 0,Y 446.418,Z 378.374,A -85,B 0,C 180,E1 -8878.7,E2 -8878.7} C_VEL
LIN {X 0,Y 446.487,Z 378.366,A -85,B 0,C 180,E1 -8881.822,E2 -8881.822} C_VEL
LIN {X 0,Y 446.461,Z 378.375,A -85,B 0,C 180,E1 -8884.848,E2 -8884.848} C_VEL
LIN {X 0,Y 446.479,Z 378.479,A -85,B 0,C 180,E1 -8887.041,E2 -8887.041} C_VEL
LIN {X 0,Y 448.252,Z 388.196,A -85,B 0,C 180,E1 -8889.343,E2 -8889.343} C_VEL
LIN {X 0,Y 447.812,Z 397.874,A -85,B 0,C 180,E1 -8891.47,E2 -8891.47} C_VEL
LIN {X 0,Y 447.64,Z 401.393,A -85,B 0,C 180,E1 -8892.232,E2 -8892.232} C_VEL
LIN {X 0,Y 451.035,Z 419.035,A -85,B 0,C 180,E1 -8892.66,E2 -8892.66} C_VEL
LIN {X 0,Y 450.234,Z 505.192,A -85,B 0,C 180,E1 -8894.044,E2 -8894.044} C_VEL
LIN {X 0,Y 449.585,Z 509.1,A -85,B 0,C 180,E1 -8894.101,E2 -8894.101} C_VEL
LIN {X 0,Y 446.705,Z 515.207,A -85,B 0,C 180,E1 -8894.157,E2 -8894.157} C_VEL
LIN {X 0,Y 443.713,Z 521.233,A -85,B 0,C 180,E1 -8894.255,E2 -8894.255} C_VEL
LIN {X 0,Y 442.904,Z 525.014,A -85,B 0,C 180,E1 -8894.383,E2 -8894.383} C_VEL
LIN {X 0,Y 442.425,Z 536.177,A -85,B 0,C 180,E1 -8894.923,E2 -8894.923} C_VEL
LIN {X 0,Y 441.887,Z 548.609,A -85,B 0,C 180,E1 -8895.729,E2 -8895.729} C_VEL
LIN {X 0,Y 441.398,Z 558.44,A -85,B 0,C 180,E1 -8896.539,E2 -8896.539} C_VEL
LIN {X 0,Y 440.765,Z 568.635,A -85,B 0,C 180,E1 -8897.569,E2 -8897.569} C_VEL
LIN {X 0,Y 440.135,Z 577.827,A -85,B 0,C 180,E1 -8898.72,E2 -8898.72} C_VEL
LIN {X 0,Y 439.537,Z 586.751,A -85,B 0,C 180,E1 -8900.103,E2 -8900.103} C_VEL
LIN {X 0,Y 439.09,Z 593.934,A -85,B 0,C 180,E1 -8901.486,E2 -8901.486} C_VEL
LIN {X 0,Y 438.79,Z 598.78,A -85,B 0,C 180,E1 -8902.638,E2 -8902.638} C_VEL
LIN {X 0,Y 438.656,Z 603.486,A -85,B 0,C 180,E1 -8904.022,E2 -8904.022} C_VEL
LIN {X 0,Y 438.409,Z 607.094,A -85,B 0,C 180,E1 -8905.403,E2 -8905.403} C_VEL
LIN {X 0,Y 438.388,Z 608.956,A -85,B 0,C 180,E1 -8906.323,E2 -8906.323} C_VEL
LIN {X 0,Y 438.39,Z 610.358,A -85,B 0,C 180,E1 -8907.243,E2 -8907.243} C_VEL
LIN {X 0,Y 438.255,Z 611.973,A -85,B 0,C 180,E1 -8909.081,E2 -8909.081} C_VEL
LIN {X 0,Y 438.229,Z 612.209,A -85,B 0,C 180,E1 -8910,E2 -8910} C_VEL
LIN {X 0,Y 438.255,Z 612.021,A -85,B 0,C 180,E1 -8910.919,E2 -8910.919} C_VEL
LIN {X 0,Y 438.39,Z 610.468,A -85,B 0,C 180,E1 -8912.757,E2 -8912.757} C_VEL
LIN {X 0,Y 438.386,Z 609.112,A -85,B 0,C 180,E1 -8913.677,E2 -8913.677} C_VEL
LIN {X 0,Y 438.474,Z 606.245,A -85,B 0,C 180,E1 -8915.058,E2 -8915.058} C_VEL
LIN {X 0,Y 438.687,Z 601.683,A -85,B 0,C 180,E1 -8916.647,E2 -8916.647} C_VEL
LIN {X 0,Y 439.005,Z 595.368,A -85,B 0,C 180,E1 -8918.284,E2 -8918.284} C_VEL
LIN {X 0,Y 439.422,Z 588.577,A -85,B 0,C 180,E1 -8919.668,E2 -8919.668} C_VEL
LIN {X 0,Y 439.953,Z 580.095,A -85,B 0,C 180,E1 -8921.052,E2 -8921.052} C_VEL
LIN {X 0,Y 440.564,Z 571.371,A -85,B 0,C 180,E1 -8922.203,E2 -8922.203} C_VEL
LIN {X 0,Y 441.196,Z 561.578,A -85,B 0,C 180,E1 -8923.259,E2 -8923.259} C_VEL
LIN {X 0,Y 441.668,Z 551.324,A -85,B 0,C 180,E1 -8924.162,E2 -8924.162} C_VEL
LIN {X 0,Y 442.299,Z 539.735,A -85,B 0,C 180,E1 -8924.964,E2 -8924.964} C_VEL
LIN {X 0,Y 442.833,Z 527.679,A -85,B 0,C 180,E1 -8925.594,E2 -8925.594} C_VEL
LIN {X 0,Y 443.257,Z 514.541,A -85,B 0,C 180,E1 -8926.08,E2 -8926.08} C_VEL
LIN {X 0,Y 443.527,Z 501.84,A -85,B 0,C 180,E1 -8926.365,E2 -8926.365} C_VEL
LIN {X 0,Y 444.2,Z 419.305,A -85,B 0,C 180,E1 -8927.708,E2 -8927.708} C_VEL
LIN {X 0,Y 440.728,Z 401.476,A -85,B 0,C 180,E1 -8928.165,E2 -8928.165} C_VEL
LIN {X 0,Y 441.335,Z 389.83,A -85,B 0,C 180,E1 -8930.752,E2 -8930.752} C_VEL
LIN {X 0,Y 439.449,Z 379.253,A -85,B 0,C 180,E1 -8933.317,E2 -8933.317} C_VEL
LIN {X 0,Y 439.432,Z 379.25,A -85,B 0,C 180,E1 -8936.604,E2 -8936.604} C_VEL
LIN {X 0,Y 439.386,Z 379.249,A -85,B 0,C 180,E1 -8939.726,E2 -8939.726} C_VEL
LIN {X 0,Y 439.377,Z 379.255,A -85,B 0,C 180,E1 -8942.946,E2 -8942.946} C_VEL
LIN {X 0,Y 439.378,Z 379.253,A -85,B 0,C 180,E1 -8946.287,E2 -8946.287} C_VEL
LIN {X 0,Y 439.405,Z 379.247,A -85,B 0,C 180,E1 -8949.849,E2 -8949.849} C_VEL
LIN {X 0,Y 439.386,Z 379.256,A -85,B 0,C 180,E1 -8952.627,E2 -8952.627} C_VEL
LIN {X 0,Y 439.41,Z 379.246,A -85,B 0,C 180,E1 -8955.272,E2 -8955.272} C_VEL
LIN {X 0,Y 439.394,Z 379.252,A -85,B 0,C 180,E1 -8958.743,E2 -8958.743} C_VEL
LIN {X 0,Y 439.389,Z 379.249,A -85,B 0,C 180,E1 -8961.606,E2 -8961.606} C_VEL
LIN {X 0,Y 439.403,Z 379.249,A -85,B 0,C 180,E1 -8964.844,E2 -8964.844} C_VEL
LIN {X 0,Y 439.378,Z 379.255,A -85,B 0,C 180,E1 -8968.14,E2 -8968.14} C_VEL
LIN {X 0,Y 439.426,Z 379.244,A -85,B 0,C 180,E1 -8971.327,E2 -8971.327} C_VEL
LIN {X 0,Y 439.403,Z 379.252,A -85,B 0,C 180,E1 -8974.415,E2 -8974.415} C_VEL
LIN {X 0,Y 439.369,Z 379.251,A -85,B 0,C 180,E1 -8977.425,E2 -8977.425} C_VEL
LIN {X 0,Y 439.447,Z 379.243,A -85,B 0,C 180,E1 -8980.663,E2 -8980.663} C_VEL
LIN {X 0,Y 439.468,Z 379.245,A -85,B 0,C 180,E1 -8984.225,E2 -8984.225} C_VEL
LIN {X 0,Y 439.489,Z 379.244,A -85,B 0,C 180,E1 -8988.001,E2 -8988.001} C_VEL
LIN {X 0,Y 439.553,Z 379.233,A -85,B 0,C 180,E1 -8991.726,E2 -8991.726} C_VEL
LIN {X 0,Y 439.627,Z 379.22,A -85,B 0,C 180,E1 -8994.496,E2 -8994.496} C_VEL
LIN {X 0,Y 439.64,Z 379.221,A -85,B 0,C 180,E1 -8998.168,E2 -8998.168} C_VEL
LIN {X 0,Y 439.768,Z 379.207,A -85,B 0,C 180,E1 -9000,E2 -9000} C_VEL
LIN {X 0,Y 439.647,Z 379.216,A -85,B 0,C 180,E1 -9002.749,E2 -9002.749} C_VEL
LIN {X 0,Y 439.618,Z 379.221,A -85,B 0,C 180,E1 -9006.425,E2 -9006.425} C_VEL
LIN {X 0,Y 439.501,Z 379.237,A -85,B 0,C 180,E1 -9009.202,E2 -9009.202} C_VEL
LIN {X 0,Y 439.509,Z 379.233,A -85,B 0,C 180,E1 -9012.726,E2 -9012.726} C_VEL
LIN {X 0,Y 439.452,Z 379.241,A -85,B 0,C 180,E1 -9016.349,E2 -9016.349} C_VEL
LIN {X 0,Y 439.408,Z 379.252,A -85,B 0,C 180,E1 -9019.626,E2 -9019.626} C_VEL
LIN {X 0,Y 439.369,Z 379.251,A -85,B 0,C 180,E1 -9022.575,E2 -9022.575} C_VEL
LIN {X 0,Y 439.402,Z 379.252,A -85,B 0,C 180,E1 -9025.585,E2 -9025.585} C_VEL
LIN {X 0,Y 439.422,Z 379.245,A -85,B 0,C 180,E1 -9028.673,E2 -9028.673} C_VEL
LIN {X 0,Y 439.373,Z 379.251,A -85,B 0,C 180,E1 -9032.03,E2 -9032.03} C_VEL
LIN {X 0,Y 439.396,Z 379.254,A -85,B 0,C 180,E1 -9035.34,E2 -9035.34} C_VEL
LIN {X 0,Y 439.381,Z 379.251,A -85,B 0,C 180,E1 -9038.595,E2 -9038.595} C_VEL
LIN {X 0,Y 439.392,Z 379.255,A -85,B 0,C 180,E1 -9041.257,E2 -9041.257} C_VEL
LIN {X 0,Y 439.409,Z 379.249,A -85,B 0,C 180,E1 -9044.728,E2 -9044.728} C_VEL
LIN {X 0,Y 439.399,Z 379.248,A -85,B 0,C 180,E1 -9047.796,E2 -9047.796} C_VEL
LIN {X 0,Y 439.433,Z 379.243,A -85,B 0,C 180,E1 -9050.228,E2 -9050.228} C_VEL
LIN {X 0,Y 439.377,Z 379.25,A -85,B 0,C 180,E1 -9053.713,E2 -9053.713} C_VEL
LIN {X 0,Y 439.376,Z 379.256,A -85,B 0,C 180,E1 -9057.054,E2 -9057.054} C_VEL
LIN {X 0,Y 439.386,Z 379.254,A -85,B 0,C 180,E1 -9060.274,E2 -9060.274} C_VEL
LIN {X 0,Y 439.445,Z 379.249,A -85,B 0,C 180,E1 -9063.541,E2 -9063.541} C_VEL
LIN {X 0,Y 440.273,Z 383.295,A -85,B 0,C 180,E1 -9064.469,E2 -9064.469} C_VEL
LIN {X 0,Y 442.082,Z 393.293,A -85,B 0,C 180,E1 -9066.582,E2 -9066.582} C_VEL
LIN {X 0,Y 441.124,Z 410.113,A -85,B 0,C 180,E1 -9069.858,E2 -9069.858} C_VEL
LIN {X 0,Y 440.555,Z 420.498,A -85,B 0,C 180,E1 -9071.865,E2 -9071.865} C_VEL
LIN {X 0,Y 444.092,Z 442.091,A -85,B 0,C 180,E1 -9072.38,E2 -9072.38} C_VEL
LIN {X 0,Y 443.288,Z 528.548,A -85,B 0,C 180,E1 -9073.803,E2 -9073.803} C_VEL
LIN {X 0,Y 442.891,Z 541.047,A -85,B 0,C 180,E1 -9074.172,E2 -9074.172} C_VEL
LIN {X 0,Y 442.302,Z 553.965,A -85,B 0,C 180,E1 -9074.741,E2 -9074.741} C_VEL
LIN {X 0,Y 441.682,Z 566.23,A -85,B 0,C 180,E1 -9075.486,E2 -9075.486} C_VEL
LIN {X 0,Y 441.007,Z 577.132,A -85,B 0,C 180,E1 -9076.342,E2 -9076.342} C_VEL
LIN {X 0,Y 440.443,Z 588.262,A -85,B 0,C 180,E1 -9077.443,E2 -9077.443} C_VEL
LIN {X 0,Y 439.908,Z 596.796,A -85,B 0,C 180,E1 -9078.48,E2 -9078.48} C_VEL
LIN {X 0,Y 439.37,Z 604.669,A -85,B 0,C 180,E1 -9079.633,E2 -9079.633} C_VEL
LIN {X 0,Y 438.932,Z 612.36,A -85,B 0,C 180,E1 -9081.018,E2 -9081.018} C_VEL
LIN {X 0,Y 438.608,Z 619.451,A -85,B 0,C 180,E1 -9082.635,E2 -9082.635} C_VEL
LIN {X 0,Y 438.397,Z 623.997,A -85,B 0,C 180,E1 -9083.963,E2 -9083.963} C_VEL
LIN {X 0,Y 438.345,Z 627.774,A -85,B 0,C 180,E1 -9085.402,E2 -9085.402} C_VEL
LIN {X 0,Y 438.26,Z 629.632,A -85,B 0,C 180,E1 -9086.322,E2 -9086.322} C_VEL
LIN {X 0,Y 438.334,Z 631.029,A -85,B 0,C 180,E1 -9087.243,E2 -9087.243} C_VEL
LIN {X 0,Y 438.23,Z 632.629,A -85,B 0,C 180,E1 -9089.081,E2 -9089.081} C_VEL
LIN {X 0,Y 438.228,Z 632.845,A -85,B 0,C 180,E1 -9090,E2 -9090} C_VEL
LIN {X 0,Y 438.278,Z 632.023,A -85,B 0,C 180,E1 -9091.838,E2 -9091.838} C_VEL
LIN {X 0,Y 438.334,Z 631.029,A -85,B 0,C 180,E1 -9092.757,E2 -9092.757} C_VEL
LIN {X 0,Y 438.259,Z 629.632,A -85,B 0,C 180,E1 -9093.678,E2 -9093.678} C_VEL
LIN {X 0,Y 438.397,Z 626.701,A -85,B 0,C 180,E1 -9095.058,E2 -9095.058} C_VEL
LIN {X 0,Y 438.448,Z 622.729,A -85,B 0,C 180,E1 -9096.442,E2 -9096.442} C_VEL
LIN {X 0,Y 438.728,Z 616.623,A -85,B 0,C 180,E1 -9098.057,E2 -9098.057} C_VEL
LIN {X 0,Y 439.058,Z 609.951,A -85,B 0,C 180,E1 -9099.443,E2 -9099.443} C_VEL
LIN {X 0,Y 439.534,Z 601.673,A -85,B 0,C 180,E1 -9100.829,E2 -9100.829} C_VEL
LIN {X 0,Y 440.123,Z 593.19,A -85,B 0,C 180,E1 -9101.981,E2 -9101.981} C_VEL
LIN {X 0,Y 440.721,Z 583.155,A -85,B 0,C 180,E1 -9103.09,E2 -9103.09} C_VEL
LIN {X 0,Y 441.299,Z 572.331,A -85,B 0,C 180,E1 -9104.056,E2 -9104.056} C_VEL
LIN {X 0,Y 441.91,Z 560.959,A -85,B 0,C 180,E1 -9104.859,E2 -9104.859} C_VEL
LIN {X 0,Y 442.526,Z 549.29,A -85,B 0,C 180,E1 -9105.486,E2 -9105.486} C_VEL
LIN {X 0,Y 443.018,Z 535.839,A -85,B 0,C 180,E1 -9106,E2 -9106} C_VEL
LIN {X 0,Y 443.418,Z 522.528,A -85,B 0,C 180,E1 -9106.31,E2 -9106.31} C_VEL
LIN {X 0,Y 444.027,Z 442.094,A -85,B 0,C 180,E1 -9107.618,E2 -9107.618} C_VEL
LIN {X 0,Y 440.526,Z 420.487,A -85,B 0,C 180,E1 -9108.131,E2 -9108.131} C_VEL
LIN {X 0,Y 441.503,Z 403.207,A -85,B 0,C 180,E1 -9111.477,E2 -9111.477} C_VEL
LIN {X 0,Y 442.09,Z 393.27,A -85,B 0,C 180,E1 -9113.418,E2 -9113.418} C_VEL
LIN {X 0,Y 440.271,Z 383.268,A -85,B 0,C 180,E1 -9115.531,E2 -9115.531} C_VEL
LIN {X 0,Y 439.438,Z 379.246,A -85,B 0,C 180,E1 -9116.412,E2 -9116.412} C_VEL
LIN {X 0,Y 439.42,Z 379.251,A -85,B 0,C 180,E1 -9118.673,E2 -9118.673} C_VEL
LIN {X 0,Y 439.373,Z 379.25,A -85,B 0,C 180,E1 -9122.031,E2 -9122.031} C_VEL
LIN {X 0,Y 439.397,Z 379.252,A -85,B 0,C 180,E1 -9125.34,E2 -9125.34} C_VEL
LIN {X 0,Y 439.385,Z 379.252,A -85,B 0,C 180,E1 -9128.595,E2 -9128.595} C_VEL
LIN {X 0,Y 439.39,Z 379.252,A -85,B 0,C 180,E1 -9131.257,E2 -9131.257} C_VEL
LIN {X 0,Y 439.404,Z 379.252,A -85,B 0,C 180,E1 -9134.729,E2 -9134.729} C_VEL
LIN {X 0,Y 439.4,Z 379.247,A -85,B 0,C 180,E1 -9137.796,E2 -9137.796} C_VEL
LIN {X 0,Y 439.432,Z 379.244,A -85,B 0,C 180,E1 -9140.228,E2 -9140.228} C_VEL
LIN {X 0,Y 439.375,Z 379.25,A -85,B 0,C 180,E1 -9143.713,E2 -9143.713} C_VEL
LIN {X 0,Y 439.374,Z 379.254,A -85,B 0,C 180,E1 -9147.054,E2 -9147.054} C_VEL
LIN {X 0,Y 439.385,Z 379.252,A -85,B 0,C 180,E1 -9150.274,E2 -9150.274} C_VEL
LIN {X 0,Y 439.431,Z 379.244,A -85,B 0,C 180,E1 -9153.396,E2 -9153.396} C_VEL
LIN {X 0,Y 439.387,Z 379.254,A -85,B 0,C 180,E1 -9156.43,E2 -9156.43} C_VEL
LIN {X 0,Y 439.391,Z 379.248,A -85,B 0,C 180,E1 -9159.397,E2 -9159.397} C_VEL
LIN {X 0,Y 439.433,Z 379.248,A -85,B 0,C 180,E1 -9162.31,E2 -9162.31} C_VEL
LIN {X 0,Y 439.45,Z 379.241,A -85,B 0,C 180,E1 -9165.174,E2 -9165.174} C_VEL
LIN {X 0,Y 439.51,Z 379.236,A -85,B 0,C 180,E1 -9168.002,E2 -9168.002} C_VEL
LIN {X 0,Y 439.507,Z 379.235,A -85,B 0,C 180,E1 -9171.726,E2 -9171.726} C_VEL
LIN {X 0,Y 439.62,Z 379.225,A -85,B 0,C 180,E1 -9174.496,E2 -9174.496} C_VEL
LIN {X 0,Y 439.637,Z 379.224,A -85,B 0,C 180,E1 -9178.168,E2 -9178.168} C_VEL
LIN {X 0,Y 439.766,Z 379.206,A -85,B 0,C 180,E1 -9180,E2 -9180} C_VEL
LIN {X 0,Y 439.659,Z 379.216,A -85,B 0,C 180,E1 -9182.749,E2 -9182.749} C_VEL
LIN {X 0,Y 439.621,Z 379.223,A -85,B 0,C 180,E1 -9186.425,E2 -9186.425} C_VEL
LIN {X 0,Y 439.501,Z 379.234,A -85,B 0,C 180,E1 -9189.202,E2 -9189.202} C_VEL
LIN {X 0,Y 439.468,Z 379.239,A -85,B 0,C 180,E1 -9192.938,E2 -9192.938} C_VEL
LIN {X 0,Y 439.45,Z 379.244,A -85,B 0,C 180,E1 -9196.349,E2 -9196.349} C_VEL
LIN {X 0,Y 439.434,Z 379.247,A -85,B 0,C 180,E1 -9199.625,E2 -9199.625} C_VEL
LIN {X 0,Y 439.369,Z 379.252,A -85,B 0,C 180,E1 -9202.575,E2 -9202.575} C_VEL
LIN {X 0,Y 439.408,Z 379.251,A -85,B 0,C 180,E1 -9205.585,E2 -9205.585} C_VEL
LIN {X 0,Y 439.424,Z 379.244,A -85,B 0,C 180,E1 -9208.673,E2 -9208.673} C_VEL
LIN {X 0,Y 439.376,Z 379.256,A -85,B 0,C 180,E1 -9211.86,E2 -9211.86} C_VEL
LIN {X 0,Y 439.403,Z 379.249,A -85,B 0,C 180,E1 -9215.156,E2 -9215.156} C_VEL
LIN {X 0,Y 439.393,Z 379.248,A -85,B 0,C 180,E1 -9218.594,E2 -9218.594} C_VEL
LIN {X 0,Y 439.392,Z 379.252,A -85,B 0,C 180,E1 -9221.257,E2 -9221.257} C_VEL
LIN {X 0,Y 439.408,Z 379.246,A -85,B 0,C 180,E1 -9224.729,E2 -9224.729} C_VEL
LIN {X 0,Y 439.398,Z 379.251,A -85,B 0,C 180,E1 -9227.796,E2 -9227.796} C_VEL
LIN {X 0,Y 439.428,Z 379.244,A -85,B 0,C 180,E1 -9230.227,E2 -9230.227} C_VEL
LIN {X 0,Y 439.38,Z 379.253,A -85,B 0,C 180,E1 -9233.713,E2 -9233.713} C_VEL
LIN {X 0,Y 439.375,Z 379.254,A -85,B 0,C 180,E1 -9237.054,E2 -9237.054} C_VEL
LIN {X 0,Y 439.385,Z 379.249,A -85,B 0,C 180,E1 -9240.274,E2 -9240.274} C_VEL
LIN {X 0,Y 439.431,Z 379.25,A -85,B 0,C 180,E1 -9243.396,E2 -9243.396} C_VEL
LIN {X 0,Y 439.434,Z 379.289,A -85,B 0,C 180,E1 -9246.807,E2 -9246.807} C_VEL
LIN {X 0,Y 441.292,Z 389.417,A -85,B 0,C 180,E1 -9249.246,E2 -9249.246} C_VEL
LIN {X 0,Y 440.828,Z 399.118,A -85,B 0,C 180,E1 -9251.406,E2 -9251.406} C_VEL
LIN {X 0,Y 440.706,Z 401.562,A -85,B 0,C 180,E1 -9251.942,E2 -9251.942} C_VEL
LIN {X 0,Y 444.292,Z 419.992,A -85,B 0,C 180,E1 -9252.401,E2 -9252.401} C_VEL
LIN {X 0,Y 443.439,Z 507.713,A -85,B 0,C 180,E1 -9253.839,E2 -9253.839} C_VEL
LIN {X 0,Y 443.013,Z 521.249,A -85,B 0,C 180,E1 -9254.236,E2 -9254.236} C_VEL
LIN {X 0,Y 442.904,Z 525.014,A -85,B 0,C 180,E1 -9254.383,E2 -9254.383} C_VEL
LIN {X 0,Y 442.032,Z 530.652,A -85,B 0,C 180,E1 -9254.612,E2 -9254.612} C_VEL
LIN {X 0,Y 437.461,Z 543.07,A -85,B 0,C 180,E1 -9255.172,E2 -9255.172} C_VEL
LIN {X 0,Y 435.224,Z 549.909,A -85,B 0,C 180,E1 -9255.591,E2 -9255.591} C_VEL
LIN {X 0,Y 434.737,Z 553.217,A -85,B 0,C 180,E1 -9255.847,E2 -9255.847} C_VEL
LIN {X 0,Y 434.137,Z 564.536,A -85,B 0,C 180,E1 -9256.901,E2 -9256.901} C_VEL
LIN {X 0,Y 433.415,Z 574.525,A -85,B 0,C 180,E1 -9258.068,E2 -9258.068} C_VEL
LIN {X 0,Y 432.723,Z 584.18,A -85,B 0,C 180,E1 -9259.472,E2 -9259.472} C_VEL
LIN {X 0,Y 432.217,Z 591.882,A -85,B 0,C 180,E1 -9260.878,E2 -9260.878} C_VEL
LIN {X 0,Y 431.739,Z 598.95,A -85,B 0,C 180,E1 -9262.517,E2 -9262.517} C_VEL
LIN {X 0,Y 431.59,Z 603.655,A -85,B 0,C 180,E1 -9263.924,E2 -9263.924} C_VEL
LIN {X 0,Y 431.339,Z 607.262,A -85,B 0,C 180,E1 -9265.327,E2 -9265.327} C_VEL
LIN {X 0,Y 431.293,Z 609.124,A -85,B 0,C 180,E1 -9266.263,E2 -9266.263} C_VEL
LIN {X 0,Y 431.32,Z 610.526,A -85,B 0,C 180,E1 -9267.198,E2 -9267.198} C_VEL
LIN {X 0,Y 431.172,Z 612.14,A -85,B 0,C 180,E1 -9269.066,E2 -9269.066} C_VEL
LIN {X 0,Y 431.145,Z 612.376,A -85,B 0,C 180,E1 -9270,E2 -9270} C_VEL
LIN {X 0,Y 431.172,Z 612.187,A -85,B 0,C 180,E1 -9270.934,E2 -9270.934} C_VEL
LIN {X 0,Y 431.32,Z 610.634,A -85,B 0,C 180,E1 -9272.802,E2 -9272.802} C_VEL
LIN {X 0,Y 431.29,Z 609.279,A -85,B 0,C 180,E1 -9273.737,E2 -9273.737} C_VEL
LIN {X 0,Y 431.42,Z 606.411,A -85,B 0,C 180,E1 -9275.141,E2 -9275.141} C_VEL
LIN {X 0,Y 431.614,Z 602.2,A -85,B 0,C 180,E1 -9276.651,E2 -9276.651} C_VEL
LIN {X 0,Y 431.871,Z 597.506,A -85,B 0,C 180,E1 -9277.951,E2 -9277.951} C_VEL
LIN {X 0,Y 432.279,Z 591.191,A -85,B 0,C 180,E1 -9279.357,E2 -9279.357} C_VEL
LIN {X 0,Y 432.821,Z 583.284,A -85,B 0,C 180,E1 -9280.762,E2 -9280.762} C_VEL
LIN {X 0,Y 433.336,Z 575.226,A -85,B 0,C 180,E1 -9281.934,E2 -9281.934} C_VEL
LIN {X 0,Y 434.027,Z 565.389,A -85,B 0,C 180,E1 -9283.103,E2 -9283.103} C_VEL
LIN {X 0,Y 434.648,Z 554.33,A -85,B 0,C 180,E1 -9284.156,E2 -9284.156} C_VEL
LIN {X 0,Y 435.259,Z 543.484,A -85,B 0,C 180,E1 -9284.972,E2 -9284.972} C_VEL
LIN {X 0,Y 435.854,Z 531.505,A -85,B 0,C 180,E1 -9285.67,E2 -9285.67} C_VEL
LIN {X 0,Y 436.34,Z 518.353,A -85,B 0,C 180,E1 -9286.222,E2 -9286.222} C_VEL
LIN {X 0,Y 436.663,Z 505.11,A -85,B 0,C 180,E1 -9286.57,E2 -9286.57} C_VEL
LIN {X 0,Y 437.474,Z 420.401,A -85,B 0,C 180,E1 -9287.973,E2 -9287.973} C_VEL
LIN {X 0,Y 433.8,Z 401.637,A -85,B 0,C 180,E1 -9288.466,E2 -9288.466} C_VEL
LIN {X 0,Y 434.386,Z 391.047,A -85,B 0,C 180,E1 -9290.851,E2 -9290.851} C_VEL
LIN {X 0,Y 432.403,Z 380.13,A -85,B 0,C 180,E1 -9293.53,E2 -9293.53} C_VEL
LIN {X 0,Y 432.395,Z 380.126,A -85,B 0,C 180,E1 -9297.072,E2 -9297.072} C_VEL
LIN {X 0,Y 432.351,Z 380.129,A -85,B 0,C 180,E1 -9300.511,E2 -9300.511} C_VEL
LIN {X 0,Y 432.363,Z 380.124,A -85,B 0,C 180,E1 -9304.004,E2 -9304.004} C_VEL
LIN {X 0,Y 432.326,Z 380.13,A -85,B 0,C 180,E1 -9307.197,E2 -9307.197} C_VEL
LIN {X 0,Y 432.337,Z 380.129,A -85,B 0,C 180,E1 -9310.179,E2 -9310.179} C_VEL
LIN {X 0,Y 432.321,Z 380.131,A -85,B 0,C 180,E1 -9313.061,E2 -9313.061} C_VEL
LIN {X 0,Y 432.345,Z 380.126,A -85,B 0,C 180,E1 -9315.664,E2 -9315.664} C_VEL
LIN {X 0,Y 432.367,Z 380.129,A -85,B 0,C 180,E1 -9318.394,E2 -9318.394} C_VEL
LIN {X 0,Y 432.351,Z 380.126,A -85,B 0,C 180,E1 -9321.851,E2 -9321.851} C_VEL
LIN {X 0,Y 432.344,Z 380.126,A -85,B 0,C 180,E1 -9325.323,E2 -9325.323} C_VEL
LIN {X 0,Y 432.327,Z 380.132,A -85,B 0,C 180,E1 -9328.654,E2 -9328.654} C_VEL
LIN {X 0,Y 432.383,Z 380.121,A -85,B 0,C 180,E1 -9331.37,E2 -9331.37} C_VEL
LIN {X 0,Y 432.366,Z 380.127,A -85,B 0,C 180,E1 -9333.968,E2 -9333.968} C_VEL
LIN {X 0,Y 432.323,Z 380.129,A -85,B 0,C 180,E1 -9337.036,E2 -9337.036} C_VEL
LIN {X 0,Y 432.397,Z 380.123,A -85,B 0,C 180,E1 -9340.513,E2 -9340.513} C_VEL
LIN {X 0,Y 432.436,Z 380.121,A -85,B 0,C 180,E1 -9343.961,E2 -9343.961} C_VEL
LIN {X 0,Y 432.464,Z 380.116,A -85,B 0,C 180,E1 -9347.803,E2 -9347.803} C_VEL
LIN {X 0,Y 432.497,Z 380.11,A -85,B 0,C 180,E1 -9351.59,E2 -9351.59} C_VEL
LIN {X 0,Y 432.603,Z 380.096,A -85,B 0,C 180,E1 -9354.406,E2 -9354.406} C_VEL
LIN {X 0,Y 432.609,Z 380.097,A -85,B 0,C 180,E1 -9358.138,E2 -9358.138} C_VEL
LIN {X 0,Y 432.738,Z 380.082,A -85,B 0,C 180,E1 -9360,E2 -9360} C_VEL
LIN {X 0,Y 432.598,Z 380.094,A -85,B 0,C 180,E1 -9362.794,E2 -9362.794} C_VEL
LIN {X 0,Y 432.568,Z 380.098,A -85,B 0,C 180,E1 -9366.53,E2 -9366.53} C_VEL
LIN {X 0,Y 432.445,Z 380.117,A -85,B 0,C 180,E1 -9369.353,E2 -9369.353} C_VEL
LIN {X 0,Y 432.45,Z 380.113,A -85,B 0,C 180,E1 -9372.812,E2 -9372.812} C_VEL
LIN {X 0,Y 432.418,Z 380.117,A -85,B 0,C 180,E1 -9376.479,E2 -9376.479} C_VEL
LIN {X 0,Y 432.344,Z 380.128,A -85,B 0,C 180,E1 -9379.96,E2 -9379.96} C_VEL
LIN {X 0,Y 432.323,Z 380.131,A -85,B 0,C 180,E1 -9382.964,E2 -9382.964} C_VEL
LIN {X 0,Y 432.365,Z 380.125,A -85,B 0,C 180,E1 -9386.032,E2 -9386.032} C_VEL
LIN {X 0,Y 432.347,Z 380.131,A -85,B 0,C 180,E1 -9389.187,E2 -9389.187} C_VEL
LIN {X 0,Y 432.326,Z 380.128,A -85,B 0,C 180,E1 -9392.443,E2 -9392.443} C_VEL
LIN {X 0,Y 432.347,Z 380.129,A -85,B 0,C 180,E1 -9395.631,E2 -9395.631} C_VEL
LIN {X 0,Y 432.344,Z 380.128,A -85,B 0,C 180,E1 -9398.714,E2 -9398.714} C_VEL
LIN {X 0,Y 432.337,Z 380.128,A -85,B 0,C 180,E1 -9401.797,E2 -9401.797} C_VEL
LIN {X 0,Y 432.344,Z 380.126,A -85,B 0,C 180,E1 -9404.346,E2 -9404.346} C_VEL
LIN {X 0,Y 432.324,Z 380.136,A -85,B 0,C 180,E1 -9407.015,E2 -9407.015} C_VEL
LIN {X 0,Y 432.34,Z 380.127,A -85,B 0,C 180,E1 -9409.82,E2 -9409.82} C_VEL
LIN {X 0,Y 432.31,Z 380.137,A -85,B 0,C 180,E1 -9413.022,E2 -9413.022} C_VEL
LIN {X 0,Y 432.363,Z 380.124,A -85,B 0,C 180,E1 -9415.996,E2 -9415.996} C_VEL
LIN {X 0,Y 432.351,Z 380.13,A -85,B 0,C 180,E1 -9419.489,E2 -9419.489} C_VEL
LIN {X 0,Y 432.394,Z 380.124,A -85,B 0,C 180,E1 -9422.928,E2 -9422.928} C_VEL
LIN {X 0,Y 432.426,Z 380.234,A -85,B 0,C 180,E1 -9423.366,E2 -9423.366} C_VEL
LIN {X 0,Y 434.727,Z 391.892,A -85,B 0,C 180,E1 -9425.908,E2 -9425.908} C_VEL
LIN {X 0,Y 435.149,Z 394.512,A -85,B 0,C 180,E1 -9426.463,E2 -9426.463} C_VEL
LIN {X 0,Y 434.201,Z 410.303,A -85,B 0,C 180,E1 -9429.592,E2 -9429.592} C_VEL
LIN {X 0,Y 433.61,Z 420.356,A -85,B 0,C 180,E1 -9431.569,E2 -9431.569} C_VEL
LIN {X 0,Y 437.338,Z 443.444,A -85,B 0,C 180,E1 -9432.125,E2 -9432.125} C_VEL
LIN {X 0,Y 436.478,Z 528.392,A -85,B 0,C 180,E1 -9433.543,E2 -9433.543} C_VEL
LIN {X 0,Y 436.079,Z 540.887,A -85,B 0,C 180,E1 -9433.918,E2 -9433.918} C_VEL
LIN {X 0,Y 435.459,Z 553.803,A -85,B 0,C 180,E1 -9434.496,E2 -9434.496} C_VEL
LIN {X 0,Y 434.787,Z 566.067,A -85,B 0,C 180,E1 -9435.251,E2 -9435.251} C_VEL
LIN {X 0,Y 434.064,Z 577.394,A -85,B 0,C 180,E1 -9436.159,E2 -9436.159} C_VEL
LIN {X 0,Y 433.479,Z 588.097,A -85,B 0,C 180,E1 -9437.238,E2 -9437.238} C_VEL
LIN {X 0,Y 432.934,Z 596.631,A -85,B 0,C 180,E1 -9438.292,E2 -9438.292} C_VEL
LIN {X 0,Y 432.352,Z 604.503,A -85,B 0,C 180,E1 -9439.463,E2 -9439.463} C_VEL
LIN {X 0,Y 431.875,Z 612.193,A -85,B 0,C 180,E1 -9440.87,E2 -9440.87} C_VEL
LIN {X 0,Y 431.541,Z 619.285,A -85,B 0,C 180,E1 -9442.514,E2 -9442.514} C_VEL
LIN {X 0,Y 431.298,Z 624.256,A -85,B 0,C 180,E1 -9444.003,E2 -9444.003} C_VEL
LIN {X 0,Y 431.275,Z 627.608,A -85,B 0,C 180,E1 -9445.326,E2 -9445.326} C_VEL
LIN {X 0,Y 431.169,Z 629.465,A -85,B 0,C 180,E1 -9446.261,E2 -9446.261} C_VEL
LIN {X 0,Y 431.228,Z 630.861,A -85,B 0,C 180,E1 -9447.197,E2 -9447.197} C_VEL
LIN {X 0,Y 431.202,Z 631.856,A -85,B 0,C 180,E1 -9448.132,E2 -9448.132} C_VEL
LIN {X 0,Y 431.143,Z 632.678,A -85,B 0,C 180,E1 -9450,E2 -9450} C_VEL
LIN {X 0,Y 431.202,Z 631.856,A -85,B 0,C 180,E1 -9451.868,E2 -9451.868} C_VEL
LIN {X 0,Y 431.228,Z 630.861,A -85,B 0,C 180,E1 -9452.802,E2 -9452.802} C_VEL
LIN {X 0,Y 431.169,Z 629.464,A -85,B 0,C 180,E1 -9453.738,E2 -9453.738} C_VEL
LIN {X 0,Y 431.309,Z 626.532,A -85,B 0,C 180,E1 -9455.142,E2 -9455.142} C_VEL
LIN {X 0,Y 431.377,Z 622.56,A -85,B 0,C 180,E1 -9456.548,E2 -9456.548} C_VEL
LIN {X 0,Y 431.681,Z 616.455,A -85,B 0,C 180,E1 -9458.19,E2 -9458.19} C_VEL
LIN {X 0,Y 432.016,Z 609.781,A -85,B 0,C 180,E1 -9459.599,E2 -9459.599} C_VEL
LIN {X 0,Y 432.543,Z 601.503,A -85,B 0,C 180,E1 -9461.006,E2 -9461.006} C_VEL
LIN {X 0,Y 433.154,Z 593.02,A -85,B 0,C 180,E1 -9462.177,E2 -9462.177} C_VEL
LIN {X 0,Y 433.748,Z 583.389,A -85,B 0,C 180,E1 -9463.263,E2 -9463.263} C_VEL
LIN {X 0,Y 434.317,Z 573.588,A -85,B 0,C 180,E1 -9464.167,E2 -9464.167} C_VEL
LIN {X 0,Y 434.926,Z 562.556,A -85,B 0,C 180,E1 -9464.984,E2 -9464.984} C_VEL
LIN {X 0,Y 435.615,Z 550.331,A -85,B 0,C 180,E1 -9465.678,E2 -9465.678} C_VEL
LIN {X 0,Y 436.134,Z 537.493,A -85,B 0,C 180,E1 -9466.199,E2 -9466.199} C_VEL
LIN {X 0,Y 436.547,Z 523.87,A -85,B 0,C 180,E1 -9466.544,E2 -9466.544} C_VEL
LIN {X 0,Y 437.283,Z 443.541,A -85,B 0,C 180,E1 -9467.872,E2 -9467.872} C_VEL
LIN {X 0,Y 433.6,Z 420.357,A -85,B 0,C 180,E1 -9468.424,E2 -9468.424} C_VEL
LIN {X 0,Y 434.612,Z 403.051,A -85,B 0,C 180,E1 -9471.834,E2 -9471.834} C_VEL
LIN {X 0,Y 435.137,Z 394.363,A -85,B 0,C 180,E1 -9473.562,E2 -9473.562} C_VEL
LIN {X 0,Y 433.014,Z 383.116,A -85,B 0,C 180,E1 -9475.99,E2 -9475.99} C_VEL
LIN {X 0,Y 432.412,Z 380.123,A -85,B 0,C 180,E1 -9476.664,E2 -9476.664} C_VEL
LIN {X 0,Y 432.345,Z 380.133,A -85,B 0,C 180,E1 -9479.187,E2 -9479.187} C_VEL
LIN {X 0,Y 432.325,Z 380.129,A -85,B 0,C 180,E1 -9482.443,E2 -9482.443} C_VEL
LIN {X 0,Y 432.346,Z 380.127,A -85,B 0,C 180,E1 -9485.632,E2 -9485.632} C_VEL
LIN {X 0,Y 432.352,Z 380.128,A -85,B 0,C 180,E1 -9489.343,E2 -9489.343} C_VEL
LIN {X 0,Y 432.335,Z 380.127,A -85,B 0,C 180,E1 -9491.797,E2 -9491.797} C_VEL
LIN {X 0,Y 432.335,Z 380.129,A -85,B 0,C 180,E1 -9494.347,E2 -9494.347} C_VEL
LIN {X 0,Y 432.327,Z 380.134,A -85,B 0,C 180,E1 -9497.015,E2 -9497.015} C_VEL
LIN {X 0,Y 432.338,Z 380.127,A -85,B 0,C 180,E1 -9499.82,E2 -9499.82} C_VEL
LIN {X 0,Y 432.308,Z 380.135,A -85,B 0,C 180,E1 -9503.022,E2 -9503.022} C_VEL
LIN {X 0,Y 432.361,Z 380.124,A -85,B 0,C 180,E1 -9505.997,E2 -9505.997} C_VEL
LIN {X 0,Y 432.35,Z 380.126,A -85,B 0,C 180,E1 -9509.49,E2 -9509.49} C_VEL
LIN {X 0,Y 432.394,Z 380.124,A -85,B 0,C 180,E1 -9512.928,E2 -9512.928} C_VEL
LIN {X 0,Y 432.37,Z 380.124,A -85,B 0,C 180,E1 -9516.023,E2 -9516.023} C_VEL
LIN {X 0,Y 432.353,Z 380.127,A -85,B 0,C 180,E1 -9519.046,E2 -9519.046} C_VEL
LIN {X 0,Y 432.38,Z 380.124,A -85,B 0,C 180,E1 -9522.011,E2 -9522.011} C_VEL
LIN {X 0,Y 432.398,Z 380.121,A -85,B 0,C 180,E1 -9524.927,E2 -9524.927} C_VEL
LIN {X 0,Y 432.483,Z 380.11,A -85,B 0,C 180,E1 -9527.804,E2 -9527.804} C_VEL
LIN {X 0,Y 432.467,Z 380.111,A -85,B 0,C 180,E1 -9531.59,E2 -9531.59} C_VEL
LIN {X 0,Y 432.597,Z 380.101,A -85,B 0,C 180,E1 -9534.406,E2 -9534.406} C_VEL
LIN {X 0,Y 432.607,Z 380.1,A -85,B 0,C 180,E1 -9538.138,E2 -9538.138} C_VEL
LIN {X 0,Y 432.735,Z 380.082,A -85,B 0,C 180,E1 -9540,E2 -9540} C_VEL
LIN {X 0,Y 432.608,Z 380.094,A -85,B 0,C 180,E1 -9542.794,E2 -9542.794} C_VEL
LIN {X 0,Y 432.576,Z 380.1,A -85,B 0,C 180,E1 -9546.53,E2 -9546.53} C_VEL
LIN {X 0,Y 432.444,Z 380.114,A -85,B 0,C 180,E1 -9549.353,E2 -9549.353} C_VEL
LIN {X 0,Y 432.433,Z 380.115,A -85,B 0,C 180,E1 -9552.804,E2 -9552.804} C_VEL
LIN {X 0,Y 432.415,Z 380.119,A -85,B 0,C 180,E1 -9556.479,E2 -9556.479} C_VEL
LIN {X 0,Y 432.376,Z 380.129,A -85,B 0,C 180,E1 -9559.959,E2 -9559.959} C_VEL
LIN {X 0,Y 432.323,Z 380.129,A -85,B 0,C 180,E1 -9562.964,E2 -9562.964} C_VEL
LIN {X 0,Y 432.368,Z 380.128,A -85,B 0,C 180,E1 -9566.032,E2 -9566.032} C_VEL
LIN {X 0,Y 432.351,Z 380.127,A -85,B 0,C 180,E1 -9569.187,E2 -9569.187} C_VEL
LIN {X 0,Y 432.327,Z 380.129,A -85,B 0,C 180,E1 -9572.293,E2 -9572.293} C_VEL
LIN {X 0,Y 432.343,Z 380.126,A -85,B 0,C 180,E1 -9574.677,E2 -9574.677} C_VEL
LIN {X 0,Y 432.35,Z 380.127,A -85,B 0,C 180,E1 -9578.149,E2 -9578.149} C_VEL
LIN {X 0,Y 432.365,Z 380.131,A -85,B 0,C 180,E1 -9581.607,E2 -9581.607} C_VEL
LIN {X 0,Y 432.343,Z 380.126,A -85,B 0,C 180,E1 -9584.346,E2 -9584.346} C_VEL
LIN {X 0,Y 432.322,Z 380.131,A -85,B 0,C 180,E1 -9587.016,E2 -9587.016} C_VEL
LIN {X 0,Y 432.335,Z 380.13,A -85,B 0,C 180,E1 -9589.821,E2 -9589.821} C_VEL
LIN {X 0,Y 432.318,Z 380.132,A -85,B 0,C 180,E1 -9593.023,E2 -9593.023} C_VEL
LIN {X 0,Y 432.362,Z 380.125,A -85,B 0,C 180,E1 -9595.996,E2 -9595.996} C_VEL
LIN {X 0,Y 432.35,Z 380.13,A -85,B 0,C 180,E1 -9599.49,E2 -9599.49} C_VEL
LIN {X 0,Y 432.394,Z 380.124,A -85,B 0,C 180,E1 -9602.928,E2 -9602.928} C_VEL
LIN {X 0,Y 432.39,Z 380.236,A -85,B 0,C 180,E1 -9606.597,E2 -9606.597} C_VEL
LIN {X 0,Y 434.341,Z 390.641,A -85,B 0,C 180,E1 -9609.147,E2 -9609.147} C_VEL
LIN {X 0,Y 433.805,Z 401.39,A -85,B 0,C 180,E1 -9611.57,E2 -9611.57} C_VEL
LIN {X 0,Y 433.793,Z 401.713,A -85,B 0,C 180,E1 -9611.642,E2 -9611.642} C_VEL
LIN {X 0,Y 437.557,Z 421.159,A -85,B 0,C 180,E1 -9612.138,E2 -9612.138} C_VEL
LIN {X 0,Y 436.639,Z 507.9,A -85,B 0,C 180,E1 -9613.58,E2 -9613.58} C_VEL
LIN {X 0,Y 436.195,Z 521.428,A -85,B 0,C 180,E1 -9613.983,E2 -9613.983} C_VEL
LIN {X 0,Y 435.696,Z 534.24,A -85,B 0,C 180,E1 -9614.565,E2 -9614.565} C_VEL
LIN {X 0,Y 435.136,Z 545.61,A -85,B 0,C 180,E1 -9615.263,E2 -9615.263} C_VEL
LIN {X 0,Y 434.737,Z 553.217,A -85,B 0,C 180,E1 -9615.847,E2 -9615.847} C_VEL
LIN {X 0,Y 433.817,Z 558.192,A -85,B 0,C 180,E1 -9616.255,E2 -9616.255} C_VEL
LIN {X 0,Y 430.555,Z 565.987,A -85,B 0,C 180,E1 -9616.942,E2 -9616.942} C_VEL
LIN {X 0,Y 427.247,Z 573.332,A -85,B 0,C 180,E1 -9617.712,E2 -9617.712} C_VEL
LIN {X 0,Y 426.246,Z 577.532,A -85,B 0,C 180,E1 -9618.257,E2 -9618.257} C_VEL
LIN {X 0,Y 425.628,Z 585.743,A -85,B 0,C 180,E1 -9619.535,E2 -9619.535} C_VEL
LIN {X 0,Y 425.108,Z 593.163,A -85,B 0,C 180,E1 -9620.964,E2 -9620.964} C_VEL
LIN {X 0,Y 424.687,Z 599.119,A -85,B 0,C 180,E1 -9622.392,E2 -9622.392} C_VEL
LIN {X 0,Y 424.512,Z 603.366,A -85,B 0,C 180,E1 -9623.668,E2 -9623.668} C_VEL
LIN {X 0,Y 424.274,Z 607.43,A -85,B 0,C 180,E1 -9625.249,E2 -9625.249} C_VEL
LIN {X 0,Y 424.199,Z 609.292,A -85,B 0,C 180,E1 -9626.2,E2 -9626.2} C_VEL
LIN {X 0,Y 424.232,Z 610.693,A -85,B 0,C 180,E1 -9627.151,E2 -9627.151} C_VEL
LIN {X 0,Y 424.092,Z 612.307,A -85,B 0,C 180,E1 -9629.051,E2 -9629.051} C_VEL
LIN {X 0,Y 424.063,Z 612.542,A -85,B 0,C 180,E1 -9630,E2 -9630} C_VEL
LIN {X 0,Y 424.092,Z 612.354,A -85,B 0,C 180,E1 -9630.95,E2 -9630.95} C_VEL
LIN {X 0,Y 424.232,Z 610.8,A -85,B 0,C 180,E1 -9632.849,E2 -9632.849} C_VEL
LIN {X 0,Y 424.196,Z 609.445,A -85,B 0,C 180,E1 -9633.8,E2 -9633.8} C_VEL
LIN {X 0,Y 424.366,Z 606.577,A -85,B 0,C 180,E1 -9635.226,E2 -9635.226} C_VEL
LIN {X 0,Y 424.542,Z 602.689,A -85,B 0,C 180,E1 -9636.655,E2 -9636.655} C_VEL
LIN {X 0,Y 424.816,Z 597.672,A -85,B 0,C 180,E1 -9638.084,E2 -9638.084} C_VEL
LIN {X 0,Y 425.272,Z 591.356,A -85,B 0,C 180,E1 -9639.513,E2 -9639.513} C_VEL
LIN {X 0,Y 425.85,Z 583.449,A -85,B 0,C 180,E1 -9640.941,E2 -9640.941} C_VEL
LIN {X 0,Y 426.385,Z 575.39,A -85,B 0,C 180,E1 -9642.132,E2 -9642.132} C_VEL
LIN {X 0,Y 427.124,Z 565.552,A -85,B 0,C 180,E1 -9643.319,E2 -9643.319} C_VEL
LIN {X 0,Y 427.748,Z 554.492,A -85,B 0,C 180,E1 -9644.389,E2 -9644.389} C_VEL
LIN {X 0,Y 428.4,Z 543.645,A -85,B 0,C 180,E1 -9645.218,E2 -9645.218} C_VEL
LIN {X 0,Y 429.042,Z 531.663,A -85,B 0,C 180,E1 -9645.925,E2 -9645.925} C_VEL
LIN {X 0,Y 429.536,Z 518.506,A -85,B 0,C 180,E1 -9646.486,E2 -9646.486} C_VEL
LIN {X 0,Y 429.864,Z 505.254,A -85,B 0,C 180,E1 -9646.84,E2 -9646.84} C_VEL
LIN {X 0,Y 430.736,Z 421.448,A -85,B 0,C 180,E1 -9648.248,E2 -9648.248} C_VEL
LIN {X 0,Y 426.876,Z 401.858,A -85,B 0,C 180,E1 -9648.762,E2 -9648.762} C_VEL
LIN {X 0,Y 427.425,Z 392.259,A -85,B 0,C 180,E1 -9650.958,E2 -9650.958} C_VEL
LIN {X 0,Y 425.335,Z 381.01,A -85,B 0,C 180,E1 -9653.783,E2 -9653.783} C_VEL
LIN {X 0,Y 425.352,Z 381.001,A -85,B 0,C 180,E1 -9657.558,E2 -9657.558} C_VEL
LIN {X 0,Y 425.291,Z 381.012,A -85,B 0,C 180,E1 -9660.816,E2 -9660.816} C_VEL
LIN {X 0,Y 425.315,Z 381.004,A -85,B 0,C 180,E1 -9664.288,E2 -9664.288} C_VEL
LIN {X 0,Y 425.282,Z 381.006,A -85,B 0,C 180,E1 -9667.694,E2 -9667.694} C_VEL
LIN {X 0,Y 425.283,Z 381.012,A -85,B 0,C 180,E1 -9670.52,E2 -9670.52} C_VEL
LIN {X 0,Y 425.261,Z 381.009,A -85,B 0,C 180,E1 -9673.351,E2 -9673.351} C_VEL
LIN {X 0,Y 425.269,Z 381.014,A -85,B 0,C 180,E1 -9676.648,E2 -9676.648} C_VEL
LIN {X 0,Y 425.299,Z 381.005,A -85,B 0,C 180,E1 -9679.874,E2 -9679.874} C_VEL
LIN {X 0,Y 425.288,Z 381.012,A -85,B 0,C 180,E1 -9682.487,E2 -9682.487} C_VEL
LIN {X 0,Y 425.312,Z 381.004,A -85,B 0,C 180,E1 -9685.817,E2 -9685.817} C_VEL
LIN {X 0,Y 425.303,Z 381.003,A -85,B 0,C 180,E1 -9689.237,E2 -9689.237} C_VEL
LIN {X 0,Y 425.354,Z 381.002,A -85,B 0,C 180,E1 -9692.443,E2 -9692.443} C_VEL
LIN {X 0,Y 425.352,Z 380.998,A -85,B 0,C 180,E1 -9695.602,E2 -9695.602} C_VEL
LIN {X 0,Y 425.298,Z 381.006,A -85,B 0,C 180,E1 -9698.682,E2 -9698.682} C_VEL
LIN {X 0,Y 425.339,Z 381.001,A -85,B 0,C 180,E1 -9701.703,E2 -9701.703} C_VEL
LIN {X 0,Y 425.354,Z 380.998,A -85,B 0,C 180,E1 -9704.671,E2 -9704.671} C_VEL
LIN {X 0,Y 425.417,Z 380.991,A -85,B 0,C 180,E1 -9707.598,E2 -9707.598} C_VEL
LIN {X 0,Y 425.447,Z 380.987,A -85,B 0,C 180,E1 -9711.45,E2 -9711.45} C_VEL
LIN {X 0,Y 425.56,Z 380.974,A -85,B 0,C 180,E1 -9714.313,E2 -9714.313} C_VEL
LIN {X 0,Y 425.579,Z 380.973,A -85,B 0,C 180,E1 -9718.107,E2 -9718.107} C_VEL
LIN {X 0,Y 425.707,Z 380.958,A -85,B 0,C 180,E1 -9720,E2 -9720} C_VEL
LIN {X 0,Y 425.552,Z 380.972,A -85,B 0,C 180,E1 -9722.84,E2 -9722.84} C_VEL
LIN {X 0,Y 425.557,Z 380.978,A -85,B 0,C 180,E1 -9725.687,E2 -9725.687} C_VEL
LIN {X 0,Y 425.413,Z 380.99,A -85,B 0,C 180,E1 -9728.551,E2 -9728.551} C_VEL
LIN {X 0,Y 425.435,Z 380.987,A -85,B 0,C 180,E1 -9732.401,E2 -9732.401} C_VEL
LIN {X 0,Y 425.393,Z 380.992,A -85,B 0,C 180,E1 -9736.312,E2 -9736.312} C_VEL
LIN {X 0,Y 425.334,Z 381.005,A -85,B 0,C 180,E1 -9739.636,E2 -9739.636} C_VEL
LIN {X 0,Y 425.31,Z 381.009,A -85,B 0,C 180,E1 -9743.365,E2 -9743.365} C_VEL
LIN {X 0,Y 425.351,Z 380.999,A -85,B 0,C 180,E1 -9746.844,E2 -9746.844} C_VEL
LIN {X 0,Y 425.295,Z 381.007,A -85,B 0,C 180,E1 -9749.719,E2 -9749.719} C_VEL
LIN {X 0,Y 425.285,Z 381.01,A -85,B 0,C 180,E1 -9753.048,E2 -9753.048} C_VEL
LIN {X 0,Y 425.285,Z 381.006,A -85,B 0,C 180,E1 -9755.928,E2 -9755.928} C_VEL
LIN {X 0,Y 425.291,Z 381.01,A -85,B 0,C 180,E1 -9759.042,E2 -9759.042} C_VEL
LIN {X 0,Y 425.281,Z 381.008,A -85,B 0,C 180,E1 -9762.652,E2 -9762.652} C_VEL
LIN {X 0,Y 425.265,Z 381.008,A -85,B 0,C 180,E1 -9766.044,E2 -9766.044} C_VEL
LIN {X 0,Y 425.278,Z 381.009,A -85,B 0,C 180,E1 -9768.621,E2 -9768.621} C_VEL
LIN {X 0,Y 425.313,Z 381.008,A -85,B 0,C 180,E1 -9771.102,E2 -9771.102} C_VEL
LIN {X 0,Y 425.303,Z 381.007,A -85,B 0,C 180,E1 -9774.664,E2 -9774.664} C_VEL
LIN {X 0,Y 425.268,Z 381.008,A -85,B 0,C 180,E1 -9778.073,E2 -9778.073} C_VEL
LIN {X 0,Y 425.334,Z 381.005,A -85,B 0,C 180,E1 -9781.368,E2 -9781.368} C_VEL
LIN {X 0,Y 425.35,Z 381.078,A -85,B 0,C 180,E1 -9783.097,E2 -9783.097} C_VEL
LIN {X 0,Y 427.733,Z 392.985,A -85,B 0,C 180,E1 -9785.746,E2 -9785.746} C_VEL
LIN {X 0,Y 428.171,Z 396.726,A -85,B 0,C 180,E1 -9786.544,E2 -9786.544} C_VEL
LIN {X 0,Y 427.063,Z 414.069,A -85,B 0,C 180,E1 -9790.033,E2 -9790.033} C_VEL
LIN {X 0,Y 426.697,Z 420.254,A -85,B 0,C 180,E1 -9791.264,E2 -9791.264} C_VEL
LIN {X 0,Y 430.573,Z 444.265,A -85,B 0,C 180,E1 -9791.851,E2 -9791.851} C_VEL
LIN {X 0,Y 429.68,Z 528.237,A -85,B 0,C 180,E1 -9793.275,E2 -9793.275} C_VEL
LIN {X 0,Y 429.257,Z 540.728,A -85,B 0,C 180,E1 -9793.656,E2 -9793.656} C_VEL
LIN {X 0,Y 428.598,Z 553.642,A -85,B 0,C 180,E1 -9794.241,E2 -9794.241} C_VEL
LIN {X 0,Y 427.918,Z 565.903,A -85,B 0,C 180,E1 -9795.008,E2 -9795.008} C_VEL
LIN {X 0,Y 427.169,Z 576.872,A -85,B 0,C 180,E1 -9795.897,E2 -9795.897} C_VEL
LIN {X 0,Y 426.521,Z 587.932,A -85,B 0,C 180,E1 -9797.026,E2 -9797.026} C_VEL
LIN {X 0,Y 425.959,Z 596.465,A -85,B 0,C 180,E1 -9798.098,E2 -9798.098} C_VEL
LIN {X 0,Y 425.327,Z 604.337,A -85,B 0,C 180,E1 -9799.287,E2 -9799.287} C_VEL
LIN {X 0,Y 424.83,Z 612.026,A -85,B 0,C 180,E1 -9800.718,E2 -9800.718} C_VEL
LIN {X 0,Y 424.461,Z 619.118,A -85,B 0,C 180,E1 -9802.388,E2 -9802.388} C_VEL
LIN {X 0,Y 424.25,Z 623.455,A -85,B 0,C 180,E1 -9803.692,E2 -9803.692} C_VEL
LIN {X 0,Y 424.205,Z 627.441,A -85,B 0,C 180,E1 -9805.248,E2 -9805.248} C_VEL
LIN {X 0,Y 424.082,Z 629.299,A -85,B 0,C 180,E1 -9806.199,E2 -9806.199} C_VEL
LIN {X 0,Y 424.123,Z 630.694,A -85,B 0,C 180,E1 -9807.15,E2 -9807.15} C_VEL
LIN {X 0,Y 424.128,Z 631.69,A -85,B 0,C 180,E1 -9808.101,E2 -9808.101} C_VEL
LIN {X 0,Y 424.061,Z 632.511,A -85,B 0,C 180,E1 -9810,E2 -9810} C_VEL
LIN {X 0,Y 424.128,Z 631.689,A -85,B 0,C 180,E1 -9811.899,E2 -9811.899} C_VEL
LIN {X 0,Y 424.123,Z 630.693,A -85,B 0,C 180,E1 -9812.849,E2 -9812.849} C_VEL
LIN {X 0,Y 424.082,Z 629.297,A -85,B 0,C 180,E1 -9813.801,E2 -9813.801} C_VEL
LIN {X 0,Y 424.222,Z 626.364,A -85,B 0,C 180,E1 -9815.228,E2 -9815.228} C_VEL
LIN {X 0,Y 424.302,Z 622.392,A -85,B 0,C 180,E1 -9816.658,E2 -9816.658} C_VEL
LIN {X 0,Y 424.613,Z 616.285,A -85,B 0,C 180,E1 -9818.327,E2 -9818.327} C_VEL
LIN {X 0,Y 424.989,Z 609.612,A -85,B 0,C 180,E1 -9819.759,E2 -9819.759} C_VEL
LIN {X 0,Y 425.529,Z 601.333,A -85,B 0,C 180,E1 -9821.19,E2 -9821.19} C_VEL
LIN {X 0,Y 426.199,Z 592.85,A -85,B 0,C 180,E1 -9822.378,E2 -9822.378} C_VEL
LIN {X 0,Y 426.871,Z 582.56,A -85,B 0,C 180,E1 -9823.548,E2 -9823.548} C_VEL
LIN {X 0,Y 427.493,Z 571.988,A -85,B 0,C 180,E1 -9824.519,E2 -9824.519} C_VEL
LIN {X 0,Y 428.196,Z 560.615,A -85,B 0,C 180,E1 -9825.347,E2 -9825.347} C_VEL
LIN {X 0,Y 428.865,Z 548.942,A -85,B 0,C 180,E1 -9825.993,E2 -9825.993} C_VEL
LIN {X 0,Y 429.413,Z 535.487,A -85,B 0,C 180,E1 -9826.521,E2 -9826.521} C_VEL
LIN {X 0,Y 429.836,Z 522.16,A -85,B 0,C 180,E1 -9826.84,E2 -9826.84} C_VEL
LIN {X 0,Y 430.429,Z 443.183,A -85,B 0,C 180,E1 -9828.169,E2 -9828.169} C_VEL
LIN {X 0,Y 426.659,Z 420.194,A -85,B 0,C 180,E1 -9828.734,E2 -9828.734} C_VEL
LIN {X 0,Y 427.654,Z 404.137,A -85,B 0,C 180,E1 -9831.954,E2 -9831.954} C_VEL
LIN {X 0,Y 428.151,Z 395.451,A -85,B 0,C 180,E1 -9833.713,E2 -9833.713} C_VEL
LIN {X 0,Y 425.994,Z 384.211,A -85,B 0,C 180,E1 -9836.188,E2 -9836.188} C_VEL
LIN {X 0,Y 425.361,Z 381.002,A -85,B 0,C 180,E1 -9836.947,E2 -9836.947} C_VEL
LIN {X 0,Y 425.293,Z 381.006,A -85,B 0,C 180,E1 -9839.719,E2 -9839.719} C_VEL
LIN {X 0,Y 425.284,Z 381.013,A -85,B 0,C 180,E1 -9843.048,E2 -9843.048} C_VEL
LIN {X 0,Y 425.284,Z 381.006,A -85,B 0,C 180,E1 -9845.929,E2 -9845.929} C_VEL
LIN {X 0,Y 425.3,Z 381.011,A -85,B 0,C 180,E1 -9849.043,E2 -9849.043} C_VEL
LIN {X 0,Y 425.277,Z 381.01,A -85,B 0,C 180,E1 -9852.653,E2 -9852.653} C_VEL
LIN {X 0,Y 425.27,Z 381.007,A -85,B 0,C 180,E1 -9856.045,E2 -9856.045} C_VEL
LIN {X 0,Y 425.278,Z 381.011,A -85,B 0,C 180,E1 -9858.622,E2 -9858.622} C_VEL
LIN {X 0,Y 425.312,Z 381.006,A -85,B 0,C 180,E1 -9861.103,E2 -9861.103} C_VEL
LIN {X 0,Y 425.301,Z 381.01,A -85,B 0,C 180,E1 -9864.664,E2 -9864.664} C_VEL
LIN {X 0,Y 425.267,Z 381.009,A -85,B 0,C 180,E1 -9868.073,E2 -9868.073} C_VEL
LIN {X 0,Y 425.333,Z 381,A -85,B 0,C 180,E1 -9871.368,E2 -9871.368} C_VEL
LIN {X 0,Y 425.356,Z 380.997,A -85,B 0,C 180,E1 -9873.506,E2 -9873.506} C_VEL
LIN {X 0,Y 425.307,Z 381.01,A -85,B 0,C 180,E1 -9876.635,E2 -9876.635} C_VEL
LIN {X 0,Y 425.331,Z 381.005,A -85,B 0,C 180,E1 -9880.364,E2 -9880.364} C_VEL
LIN {X 0,Y 425.391,Z 380.993,A -85,B 0,C 180,E1 -9883.688,E2 -9883.688} C_VEL
LIN {X 0,Y 425.433,Z 380.987,A -85,B 0,C 180,E1 -9887.599,E2 -9887.599} C_VEL
LIN {X 0,Y 425.411,Z 380.99,A -85,B 0,C 180,E1 -9891.449,E2 -9891.449} C_VEL
LIN {X 0,Y 425.553,Z 380.98,A -85,B 0,C 180,E1 -9894.313,E2 -9894.313} C_VEL
LIN {X 0,Y 425.576,Z 380.975,A -85,B 0,C 180,E1 -9898.107,E2 -9898.107} C_VEL
LIN {X 0,Y 425.705,Z 380.958,A -85,B 0,C 180,E1 -9900,E2 -9900} C_VEL
LIN {X 0,Y 425.56,Z 380.972,A -85,B 0,C 180,E1 -9902.84,E2 -9902.84} C_VEL
LIN {X 0,Y 425.534,Z 380.976,A -85,B 0,C 180,E1 -9906.639,E2 -9906.639} C_VEL
LIN {X 0,Y 425.403,Z 380.992,A -85,B 0,C 180,E1 -9909.509,E2 -9909.509} C_VEL
LIN {X 0,Y 425.396,Z 380.992,A -85,B 0,C 180,E1 -9912.904,E2 -9912.904} C_VEL
LIN {X 0,Y 425.364,Z 380.996,A -85,B 0,C 180,E1 -9916.605,E2 -9916.605} C_VEL
LIN {X 0,Y 425.364,Z 381,A -85,B 0,C 180,E1 -9919.648,E2 -9919.648} C_VEL
LIN {X 0,Y 425.31,Z 381.004,A -85,B 0,C 180,E1 -9923.365,E2 -9923.365} C_VEL
LIN {X 0,Y 425.351,Z 380.997,A -85,B 0,C 180,E1 -9926.845,E2 -9926.845} C_VEL
LIN {X 0,Y 425.318,Z 381.009,A -85,B 0,C 180,E1 -9929.718,E2 -9929.718} C_VEL
LIN {X 0,Y 425.284,Z 381.006,A -85,B 0,C 180,E1 -9933.048,E2 -9933.048} C_VEL
LIN {X 0,Y 425.287,Z 381.009,A -85,B 0,C 180,E1 -9935.929,E2 -9935.929} C_VEL
LIN {X 0,Y 425.306,Z 381.004,A -85,B 0,C 180,E1 -9939.045,E2 -9939.045} C_VEL
LIN {X 0,Y 425.294,Z 381.007,A -85,B 0,C 180,E1 -9941.959,E2 -9941.959} C_VEL
LIN {X 0,Y 425.288,Z 381.01,A -85,B 0,C 180,E1 -9945.283,E2 -9945.283} C_VEL
LIN {X 0,Y 425.276,Z 381.007,A -85,B 0,C 180,E1 -9948.622,E2 -9948.622} C_VEL
LIN {X 0,Y 425.312,Z 381.006,A -85,B 0,C 180,E1 -9951.103,E2 -9951.103} C_VEL
LIN {X 0,Y 425.303,Z 381.004,A -85,B 0,C 180,E1 -9954.664,E2 -9954.664} C_VEL
LIN {X 0,Y 425.267,Z 381.008,A -85,B 0,C 180,E1 -9958.073,E2 -9958.073} C_VEL
LIN {X 0,Y 425.334,Z 381.006,A -85,B 0,C 180,E1 -9961.368,E2 -9961.368} C_VEL
LIN {X 0,Y 425.298,Z 381.009,A -85,B 0,C 180,E1 -9964.555,E2 -9964.555} C_VEL
LIN {X 0,Y 425.363,Z 381.181,A -85,B 0,C 180,E1 -9966.38,E2 -9966.38} C_VEL
LIN {X 0,Y 427.376,Z 391.842,A -85,B 0,C 180,E1 -9969.037,E2 -9969.037} C_VEL
LIN {X 0,Y 427,Z 399.442,A -85,B 0,C 180,E1 -9970.781,E2 -9970.781} C_VEL
LIN {X 0,Y 426.884,Z 401.85,A -85,B 0,C 180,E1 -9971.328,E2 -9971.328} C_VEL
LIN {X 0,Y 430.782,Z 421.835,A -85,B 0,C 180,E1 -9971.856,E2 -9971.856} C_VEL
LIN {X 0,Y 429.851,Z 508.087,A -85,B 0,C 180,E1 -9973.313,E2 -9973.313} C_VEL
LIN {X 0,Y 429.394,Z 521.606,A -85,B 0,C 180,E1 -9973.723,E2 -9973.723} C_VEL
LIN {X 0,Y 428.849,Z 534.416,A -85,B 0,C 180,E1 -9974.312,E2 -9974.312} C_VEL
LIN {X 0,Y 428.279,Z 545.783,A -85,B 0,C 180,E1 -9975.022,E2 -9975.022} C_VEL
LIN {X 0,Y 427.706,Z 556.531,A -85,B 0,C 180,E1 -9975.887,E2 -9975.887} C_VEL
LIN {X 0,Y 426.976,Z 567.917,A -85,B 0,C 180,E1 -9977.04,E2 -9977.04} C_VEL
LIN {X 0,Y 426.246,Z 577.532,A -85,B 0,C 180,E1 -9978.257,E2 -9978.257} C_VEL
LIN {X 0,Y 425.268,Z 581.554,A -85,B 0,C 180,E1 -9978.827,E2 -9978.827} C_VEL
LIN {X 0,Y 420.578,Z 589.998,A -85,B 0,C 180,E1 -9980.18,E2 -9980.18} C_VEL
LIN {X 0,Y 418.343,Z 594.321,A -85,B 0,C 180,E1 -9981.035,E2 -9981.035} C_VEL
LIN {X 0,Y 417.861,Z 596.306,A -85,B 0,C 180,E1 -9981.496,E2 -9981.496} C_VEL
LIN {X 0,Y 417.48,Z 602.575,A -85,B 0,C 180,E1 -9983.233,E2 -9983.233} C_VEL
LIN {X 0,Y 417.315,Z 606.533,A -85,B 0,C 180,E1 -9984.685,E2 -9984.685} C_VEL
LIN {X 0,Y 417.109,Z 609.46,A -85,B 0,C 180,E1 -9986.136,E2 -9986.136} C_VEL
LIN {X 0,Y 417.133,Z 610.861,A -85,B 0,C 180,E1 -9987.103,E2 -9987.103} C_VEL
LIN {X 0,Y 417.081,Z 611.859,A -85,B 0,C 180,E1 -9988.069,E2 -9988.069} C_VEL
LIN {X 0,Y 416.984,Z 612.709,A -85,B 0,C 180,E1 -9990,E2 -9990} C_VEL
LIN {X 0,Y 417.014,Z 612.52,A -85,B 0,C 180,E1 -9990.966,E2 -9990.966} C_VEL
LIN {X 0,Y 417.081,Z 611.935,A -85,B 0,C 180,E1 -9991.931,E2 -9991.931} C_VEL
LIN {X 0,Y 417.132,Z 610.967,A -85,B 0,C 180,E1 -9992.897,E2 -9992.897} C_VEL
LIN {X 0,Y 417.105,Z 609.612,A -85,B 0,C 180,E1 -9993.865,E2 -9993.865} C_VEL
LIN {X 0,Y 417.312,Z 606.743,A -85,B 0,C 180,E1 -9995.315,E2 -9995.315} C_VEL
LIN {X 0,Y 417.48,Z 602.855,A -85,B 0,C 180,E1 -9996.768,E2 -9996.768} C_VEL
LIN {X 0,Y 417.786,Z 597.838,A -85,B 0,C 180,E1 -9998.221,E2 -9998.221} C_VEL
LIN {X 0,Y 418.259,Z 591.521,A -85,B 0,C 180,E1 -9999.674,E2 -9999.674} C_VEL
LIN {X 0,Y 418.865,Z 583.614,A -85,B 0,C 180,E1 -10001.126,E2 -10001.126} C_VEL
LIN {X 0,Y 419.453,Z 575.553,A -85,B 0,C 180,E1 -10002.335,E2 -10002.335} C_VEL
LIN {X 0,Y 420.212,Z 565.715,A -85,B 0,C 180,E1 -10003.542,E2 -10003.542} C_VEL
LIN {X 0,Y 420.87,Z 554.654,A -85,B 0,C 180,E1 -10004.63,E2 -10004.63} C_VEL
LIN {X 0,Y 421.562,Z 543.805,A -85,B 0,C 180,E1 -10005.471,E2 -10005.471} C_VEL
LIN {X 0,Y 422.232,Z 531.822,A -85,B 0,C 180,E1 -10006.189,E2 -10006.189} C_VEL
LIN {X 0,Y 422.734,Z 518.659,A -85,B 0,C 180,E1 -10006.759,E2 -10006.759} C_VEL
LIN {X 0,Y 423.098,Z 505.398,A -85,B 0,C 180,E1 -10007.117,E2 -10007.117} C_VEL
LIN {X 0,Y 423.934,Z 421.807,A -85,B 0,C 180,E1 -10008.548,E2 -10008.548} C_VEL
LIN {X 0,Y 419.987,Z 402.009,A -85,B 0,C 180,E1 -10009.085,E2 -10009.085} C_VEL
LIN {X 0,Y 420.476,Z 393.723,A -85,B 0,C 180,E1 -10011.01,E2 -10011.01} C_VEL
LIN {X 0,Y 418.302,Z 381.887,A -85,B 0,C 180,E1 -10014.011,E2 -10014.011} C_VEL
LIN {X 0,Y 418.314,Z 381.88,A -85,B 0,C 180,E1 -10017.071,E2 -10017.071} C_VEL
LIN {X 0,Y 418.248,Z 381.884,A -85,B 0,C 180,E1 -10020.272,E2 -10020.272} C_VEL
LIN {X 0,Y 418.252,Z 381.882,A -85,B 0,C 180,E1 -10023.677,E2 -10023.677} C_VEL
LIN {X 0,Y 418.244,Z 381.884,A -85,B 0,C 180,E1 -10027.224,E2 -10027.224} C_VEL
LIN {X 0,Y 418.25,Z 381.882,A -85,B 0,C 180,E1 -10029.683,E2 -10029.683} C_VEL
LIN {X 0,Y 418.233,Z 381.888,A -85,B 0,C 180,E1 -10032.321,E2 -10032.321} C_VEL
LIN {X 0,Y 418.243,Z 381.884,A -85,B 0,C 180,E1 -10035.109,E2 -10035.109} C_VEL
LIN {X 0,Y 418.247,Z 381.883,A -85,B 0,C 180,E1 -10037.767,E2 -10037.767} C_VEL
LIN {X 0,Y 418.264,Z 381.886,A -85,B 0,C 180,E1 -10040.618,E2 -10040.618} C_VEL
LIN {X 0,Y 418.249,Z 381.884,A -85,B 0,C 180,E1 -10043.976,E2 -10043.976} C_VEL
LIN {X 0,Y 418.262,Z 381.881,A -85,B 0,C 180,E1 -10047.156,E2 -10047.156} C_VEL
LIN {X 0,Y 418.276,Z 381.88,A -85,B 0,C 180,E1 -10050.839,E2 -10050.839} C_VEL
LIN {X 0,Y 418.273,Z 381.884,A -85,B 0,C 180,E1 -10054.096,E2 -10054.096} C_VEL
LIN {X 0,Y 418.242,Z 381.883,A -85,B 0,C 180,E1 -10057.264,E2 -10057.264} C_VEL
LIN {X 0,Y 418.321,Z 381.878,A -85,B 0,C 180,E1 -10060.366,E2 -10060.366} C_VEL
LIN {X 0,Y 418.322,Z 381.873,A -85,B 0,C 180,E1 -10063.405,E2 -10063.405} C_VEL
LIN {X 0,Y 418.351,Z 381.869,A -85,B 0,C 180,E1 -10066.999,E2 -10066.999} C_VEL
LIN {X 0,Y 418.345,Z 381.873,A -85,B 0,C 180,E1 -10070.329,E2 -10070.329} C_VEL
LIN {X 0,Y 418.518,Z 381.852,A -85,B 0,C 180,E1 -10072.279,E2 -10072.279} C_VEL
LIN {X 0,Y 418.519,Z 381.852,A -85,B 0,C 180,E1 -10074.217,E2 -10074.217} C_VEL
LIN {X 0,Y 418.548,Z 381.849,A -85,B 0,C 180,E1 -10078.075,E2 -10078.075} C_VEL
LIN {X 0,Y 418.676,Z 381.834,A -85,B 0,C 180,E1 -10080,E2 -10080} C_VEL
LIN {X 0,Y 418.507,Z 381.85,A -85,B 0,C 180,E1 -10082.888,E2 -10082.888} C_VEL
LIN {X 0,Y 418.516,Z 381.856,A -85,B 0,C 180,E1 -10085.783,E2 -10085.783} C_VEL
LIN {X 0,Y 418.383,Z 381.865,A -85,B 0,C 180,E1 -10088.695,E2 -10088.695} C_VEL
LIN {X 0,Y 418.336,Z 381.879,A -85,B 0,C 180,E1 -10091.63,E2 -10091.63} C_VEL
LIN {X 0,Y 418.311,Z 381.874,A -85,B 0,C 180,E1 -10094.597,E2 -10094.597} C_VEL
LIN {X 0,Y 418.293,Z 381.883,A -85,B 0,C 180,E1 -10097.604,E2 -10097.604} C_VEL
LIN {X 0,Y 418.255,Z 381.881,A -85,B 0,C 180,E1 -10100.663,E2 -10100.663} C_VEL
LIN {X 0,Y 418.29,Z 381.88,A -85,B 0,C 180,E1 -10103.781,E2 -10103.781} C_VEL
LIN {X 0,Y 418.314,Z 381.877,A -85,B 0,C 180,E1 -10107.07,E2 -10107.07} C_VEL
LIN {X 0,Y 418.249,Z 381.882,A -85,B 0,C 180,E1 -10110.272,E2 -10110.272} C_VEL
LIN {X 0,Y 418.251,Z 381.885,A -85,B 0,C 180,E1 -10113.677,E2 -10113.677} C_VEL
LIN {X 0,Y 418.243,Z 381.89,A -85,B 0,C 180,E1 -10117.224,E2 -10117.224} C_VEL
LIN {X 0,Y 418.25,Z 381.884,A -85,B 0,C 180,E1 -10119.682,E2 -10119.682} C_VEL
LIN {X 0,Y 418.235,Z 381.884,A -85,B 0,C 180,E1 -10122.321,E2 -10122.321} C_VEL
LIN {X 0,Y 418.242,Z 381.89,A -85,B 0,C 180,E1 -10125.109,E2 -10125.109} C_VEL
LIN {X 0,Y 418.243,Z 381.883,A -85,B 0,C 180,E1 -10127.767,E2 -10127.767} C_VEL
LIN {X 0,Y 418.259,Z 381.883,A -85,B 0,C 180,E1 -10130.619,E2 -10130.619} C_VEL
LIN {X 0,Y 418.247,Z 381.882,A -85,B 0,C 180,E1 -10133.976,E2 -10133.976} C_VEL
LIN {X 0,Y 418.261,Z 381.885,A -85,B 0,C 180,E1 -10137.156,E2 -10137.156} C_VEL
LIN {X 0,Y 418.272,Z 381.887,A -85,B 0,C 180,E1 -10140.895,E2 -10140.895} C_VEL
